KUKA KRL program: EPS_2_26115_ST7262_A_20260223020031.src

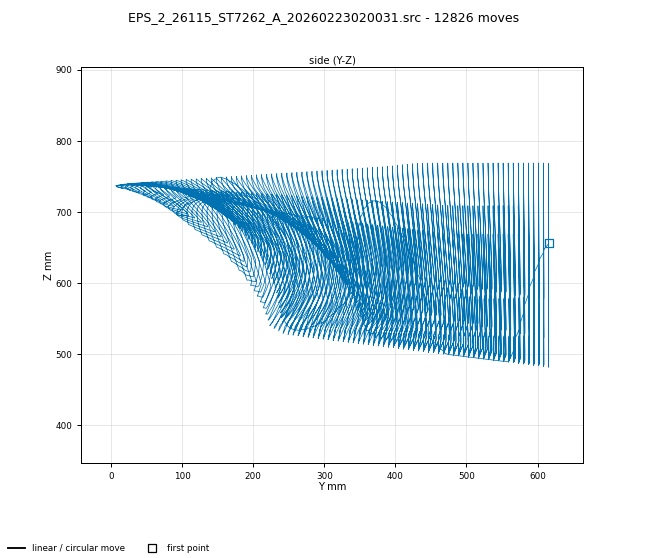
[picture p0: tool path of EPS_2_26115_ST7262_A_20260223020031.src, 12826 of 12828 moves have a stored position in this frame; points joined in program order, loops and branches not executed]
&ACCESS RVP
&REL 4
&COMMENT QRS 19112012
&PARAM EDITMASK = *
DEF PART()
EXT BAS (BAS_COMMAND :IN,REAL :IN )
INT I
BAS (#INITMOV,0 )

;KUKA QRS Post kuka4.cps  Date:22-06-2017 !

File_ID=3072

QRS_PRE_INIT()

;Init var - Until changes are made in qrs_pre_init
Outlet_Square_prg=0
Inlet_1_Square_prg=0
Inlet_2_Square_prg=0
Inlet_3_Square_prg=0
Inlet_4_Square_prg=0
Inlet_5_Square_prg=0

Outlet_1={X 0.000, Y 435.000, Z 586.000, B 0.000, E1 0.000 }
Inlet_1={X 0.000, Y 481.370, Z 486.000, B 0.000, E1 90.000 }
Inlet_2={X 0.000, Y 478.250, Z 526.000, B 0.000, E1 195.000 }
Outlet_1_type=366
Inlet_1_type=366
Inlet_2_type=366
;QRS#1=Sidecore dimensions
;QRS#2=375-15" PVC SDR 35 Cut Back
;QRS#3=375-15" PVC SDR 35
;QRS#4=375-15" PVC SDR 35
;QRS#5=
;QRS#6=
;QRS#7=
;QRS#8=
;QRS#9=20Y PSX
;QRS#10=20Y PSX
;QRS#11=20Y PSX
;QRS#12=
;QRS#13=
;QRS#14=
;QRS#15=
;QRS#16=1220x127x1067 3,5'
;QRS#17=EPS Height
;QRS#18=769
;QRS#19=*
;QRS#20= UPDATED VERSION 22-06-2017
;QRS#21=*
Outlet_Square=0250
Inlet_1_Square=0250
Inlet_2_Square=0250
Inlet_3_Square=0
Inlet_4_Square=0
Inlet_5_Square=0
Mill_Square=1
Outlet_Square_Prg=275
Inlet_1_Square_prg=252
Inlet_2_Square_prg=252

QRS_INIT()

$ADVANCE=5

; T1
PTP {E1 173.417,E2 173.417}
PTP {X 0,Y 615.494,A -85,B 0,C 180,E1 173.417,E2 173.417,E3 0,E4 0,E5 0,E6 0}
QRS_SPEED_INIT()
LIN {X 0,Y 615.494,Z 656.327,A -85,B 0,C 180,E1 173.417,E2 173.417,E3 0,E4 0,E5 0,E6 0} C_VEL
LIN {X 0,Y 615.488,Z 650.936,A -85,B 0,C 180,E1 172.124,E2 172.124} C_VEL
LIN {X 0,Y 615.489,Z 644.145,A -85,B 0,C 180,E1 170.801,E2 170.801} C_VEL
LIN {X 0,Y 615.492,Z 635.981,A -85,B 0,C 180,E1 169.473,E2 169.473} C_VEL
LIN {X 0,Y 615.494,Z 626.246,A -85,B 0,C 180,E1 168.139,E2 168.139} C_VEL
LIN {X 0,Y 615.49,Z 616.219,A -85,B 0,C 180,E1 166.966,E2 166.966} C_VEL
LIN {X 0,Y 615.496,Z 604.053,A -85,B 0,C 180,E1 165.759,E2 165.759} C_VEL
LIN {X 0,Y 615.5,Z 590.268,A -85,B 0,C 180,E1 164.604,E2 164.604} C_VEL
LIN {X 0,Y 615.495,Z 575.471,A -85,B 0,C 180,E1 163.567,E2 163.567} C_VEL
LIN {X 0,Y 615.499,Z 561.122,A -85,B 0,C 180,E1 162.73,E2 162.73} C_VEL
LIN {X 0,Y 615.48,Z 547.09,A -85,B 0,C 180,E1 162.043,E2 162.043} C_VEL
LIN {X 0,Y 615.499,Z 531.957,A -85,B 0,C 180,E1 161.434,E2 161.434} C_VEL
LIN {X 0,Y 615.48,Z 515.455,A -85,B 0,C 180,E1 160.921,E2 160.921} C_VEL
LIN {X 0,Y 615.494,Z 498.994,A -85,B 0,C 180,E1 160.554,E2 160.554} C_VEL
LIN {X 0,Y 615.49,Z 482.974,A -85,B 0,C 180,E1 160.315,E2 160.315} C_VEL
LIN {X 0,Y 615.487,Z 482.007,A -85,B 0,C 180,E1 159.269,E2 159.269} C_VEL
LIN {X 0,Y 615.491,Z 482.006,A -85,B 0,C 180,E1 156.443,E2 156.443} C_VEL
LIN {X 0,Y 615.479,Z 482.009,A -85,B 0,C 180,E1 153.555,E2 153.555} C_VEL
LIN {X 0,Y 615.491,Z 482.009,A -85,B 0,C 180,E1 151.342,E2 151.342} C_VEL
LIN {X 0,Y 615.477,Z 482.007,A -85,B 0,C 180,E1 148.916,E2 148.916} C_VEL
LIN {X 0,Y 615.494,Z 482.006,A -85,B 0,C 180,E1 146.465,E2 146.465} C_VEL
LIN {X 0,Y 615.481,Z 482.008,A -85,B 0,C 180,E1 143.574,E2 143.574} C_VEL
LIN {X 0,Y 615.49,Z 482.011,A -85,B 0,C 180,E1 140.938,E2 140.938} C_VEL
LIN {X 0,Y 615.482,Z 482.01,A -85,B 0,C 180,E1 138.525,E2 138.525} C_VEL
LIN {X 0,Y 615.482,Z 482.007,A -85,B 0,C 180,E1 135.849,E2 135.849} C_VEL
LIN {X 0,Y 615.485,Z 482.006,A -85,B 0,C 180,E1 133.047,E2 133.047} C_VEL
LIN {X 0,Y 615.495,Z 482.005,A -85,B 0,C 180,E1 130.089,E2 130.089} C_VEL
LIN {X 0,Y 615.49,Z 482.006,A -85,B 0,C 180,E1 127.242,E2 127.242} C_VEL
LIN {X 0,Y 615.477,Z 482.007,A -85,B 0,C 180,E1 124.698,E2 124.698} C_VEL
LIN {X 0,Y 615.497,Z 482.008,A -85,B 0,C 180,E1 122.332,E2 122.332} C_VEL
LIN {X 0,Y 615.485,Z 482.01,A -85,B 0,C 180,E1 119.407,E2 119.407} C_VEL
LIN {X 0,Y 615.492,Z 482.008,A -85,B 0,C 180,E1 117.045,E2 117.045} C_VEL
LIN {X 0,Y 615.498,Z 482.03,A -85,B 0,C 180,E1 114.141,E2 114.141} C_VEL
LIN {X 0,Y 615.499,Z 487.086,A -85,B 0,C 180,E1 111.432,E2 111.432} C_VEL
LIN {X 0,Y 615.477,Z 492.467,A -85,B 0,C 180,E1 108.6,E2 108.6} C_VEL
LIN {X 0,Y 615.494,Z 497.748,A -85,B 0,C 180,E1 105.906,E2 105.906} C_VEL
LIN {X 0,Y 615.487,Z 503.194,A -85,B 0,C 180,E1 103.202,E2 103.202} C_VEL
LIN {X 0,Y 615.476,Z 508.733,A -85,B 0,C 180,E1 100.528,E2 100.528} C_VEL
LIN {X 0,Y 615.487,Z 514.32,A -85,B 0,C 180,E1 97.876,E2 97.876} C_VEL
LIN {X 0,Y 615.491,Z 520.717,A -85,B 0,C 180,E1 94.913,E2 94.913} C_VEL
LIN {X 0,Y 615.481,Z 521.339,A -85,B 0,C 180,E1 94.626,E2 94.626} C_VEL
LIN {X 0,Y 615.497,Z 540.982,A -85,B 0,C 180,E1 94.319,E2 94.319} C_VEL
LIN {X 0,Y 615.486,Z 557.536,A -85,B 0,C 180,E1 93.929,E2 93.929} C_VEL
LIN {X 0,Y 615.475,Z 573.048,A -85,B 0,C 180,E1 93.438,E2 93.438} C_VEL
LIN {X 0,Y 615.487,Z 589.037,A -85,B 0,C 180,E1 92.782,E2 92.782} C_VEL
LIN {X 0,Y 615.498,Z 603.591,A -85,B 0,C 180,E1 92.046,E2 92.046} C_VEL
LIN {X 0,Y 615.497,Z 618.433,A -85,B 0,C 180,E1 91.146,E2 91.146} C_VEL
LIN {X 0,Y 615.497,Z 632.037,A -85,B 0,C 180,E1 90.164,E2 90.164} C_VEL
LIN {X 0,Y 615.494,Z 643.706,A -85,B 0,C 180,E1 89.183,E2 89.183} C_VEL
LIN {X 0,Y 615.499,Z 655.309,A -85,B 0,C 180,E1 88.038,E2 88.038} C_VEL
LIN {X 0,Y 615.492,Z 666.597,A -85,B 0,C 180,E1 86.728,E2 86.728} C_VEL
LIN {X 0,Y 615.491,Z 676.122,A -85,B 0,C 180,E1 85.416,E2 85.416} C_VEL
LIN {X 0,Y 615.493,Z 684.181,A -85,B 0,C 180,E1 84.102,E2 84.102} C_VEL
LIN {X 0,Y 615.493,Z 690.938,A -85,B 0,C 180,E1 82.785,E2 82.785} C_VEL
LIN {X 0,Y 615.487,Z 696.437,A -85,B 0,C 180,E1 81.464,E2 81.464} C_VEL
LIN {X 0,Y 615.496,Z 700.913,A -85,B 0,C 180,E1 80.139,E2 80.139} C_VEL
LIN {X 0,Y 615.494,Z 704.24,A -85,B 0,C 180,E1 78.808,E2 78.808} C_VEL
LIN {X 0,Y 615.489,Z 706.639,A -85,B 0,C 180,E1 77.471,E2 77.471} C_VEL
LIN {X 0,Y 615.49,Z 708.009,A -85,B 0,C 180,E1 76.068,E2 76.068} C_VEL
LIN {X 0,Y 615.492,Z 708.351,A -85,B 0,C 180,E1 74.775,E2 74.775} C_VEL
LIN {X 0,Y 615.491,Z 707.707,A -85,B 0,C 180,E1 73.414,E2 73.414} C_VEL
LIN {X 0,Y 615.489,Z 706.012,A -85,B 0,C 180,E1 72.044,E2 72.044} C_VEL
LIN {X 0,Y 615.49,Z 703.29,A -85,B 0,C 180,E1 70.663,E2 70.663} C_VEL
LIN {X 0,Y 615.497,Z 698.197,A -85,B 0,C 180,E1 68.92,E2 68.92} C_VEL
LIN {X 0,Y 615.499,Z 692.193,A -85,B 0,C 180,E1 67.406,E2 67.406} C_VEL
LIN {X 0,Y 615.492,Z 685.183,A -85,B 0,C 180,E1 65.992,E2 65.992} C_VEL
LIN {X 0,Y 615.493,Z 677.649,A -85,B 0,C 180,E1 64.721,E2 64.721} C_VEL
LIN {X 0,Y 615.492,Z 668.374,A -85,B 0,C 180,E1 63.407,E2 63.407} C_VEL
LIN {X 0,Y 615.493,Z 658.93,A -85,B 0,C 180,E1 62.271,E2 62.271} C_VEL
LIN {X 0,Y 615.494,Z 648.24,A -85,B 0,C 180,E1 61.157,E2 61.157} C_VEL
LIN {X 0,Y 615.495,Z 636.643,A -85,B 0,C 180,E1 60.114,E2 60.114} C_VEL
LIN {X 0,Y 615.496,Z 623.154,A -85,B 0,C 180,E1 59.082,E2 59.082} C_VEL
LIN {X 0,Y 615.498,Z 610.049,A -85,B 0,C 180,E1 58.236,E2 58.236} C_VEL
LIN {X 0,Y 615.498,Z 595.659,A -85,B 0,C 180,E1 57.447,E2 57.447} C_VEL
LIN {X 0,Y 615.483,Z 580.647,A -85,B 0,C 180,E1 56.765,E2 56.765} C_VEL
LIN {X 0,Y 615.477,Z 565.676,A -85,B 0,C 180,E1 56.224,E2 56.224} C_VEL
LIN {X 0,Y 615.489,Z 551.02,A -85,B 0,C 180,E1 55.81,E2 55.81} C_VEL
LIN {X 0,Y 615.492,Z 535.775,A -85,B 0,C 180,E1 55.493,E2 55.493} C_VEL
LIN {X 0,Y 615.48,Z 521.345,A -85,B 0,C 180,E1 55.287,E2 55.287} C_VEL
LIN {X 0,Y 615.491,Z 515.876,A -85,B 0,C 180,E1 52.76,E2 52.76} C_VEL
LIN {X 0,Y 615.489,Z 509.829,A -85,B 0,C 180,E1 49.911,E2 49.911} C_VEL
LIN {X 0,Y 615.49,Z 505.13,A -85,B 0,C 180,E1 47.649,E2 47.649} C_VEL
LIN {X 0,Y 615.48,Z 499.601,A -85,B 0,C 180,E1 44.932,E2 44.932} C_VEL
LIN {X 0,Y 615.494,Z 493.965,A -85,B 0,C 180,E1 42.083,E2 42.083} C_VEL
LIN {X 0,Y 615.498,Z 489.481,A -85,B 0,C 180,E1 39.75,E2 39.75} C_VEL
LIN {X 0,Y 615.48,Z 484.243,A -85,B 0,C 180,E1 36.938,E2 36.938} C_VEL
LIN {X 0,Y 615.495,Z 482.008,A -85,B 0,C 180,E1 35.726,E2 35.726} C_VEL
LIN {X 0,Y 615.491,Z 482.014,A -85,B 0,C 180,E1 33.236,E2 33.236} C_VEL
LIN {X 0,Y 615.483,Z 482.009,A -85,B 0,C 180,E1 30.92,E2 30.92} C_VEL
LIN {X 0,Y 615.483,Z 482.007,A -85,B 0,C 180,E1 28.452,E2 28.452} C_VEL
LIN {X 0,Y 615.496,Z 482.005,A -85,B 0,C 180,E1 25.574,E2 25.574} C_VEL
LIN {X 0,Y 615.482,Z 482.008,A -85,B 0,C 180,E1 22.845,E2 22.845} C_VEL
LIN {X 0,Y 615.477,Z 482.01,A -85,B 0,C 180,E1 20.033,E2 20.033} C_VEL
LIN {X 0,Y 615.49,Z 482.008,A -85,B 0,C 180,E1 17.271,E2 17.271} C_VEL
LIN {X 0,Y 615.493,Z 482.008,A -85,B 0,C 180,E1 14.549,E2 14.549} C_VEL
LIN {X 0,Y 615.48,Z 482.01,A -85,B 0,C 180,E1 11.861,E2 11.861} C_VEL
LIN {X 0,Y 615.488,Z 482.008,A -85,B 0,C 180,E1 9.199,E2 9.199} C_VEL
LIN {X 0,Y 615.491,Z 482.006,A -85,B 0,C 180,E1 6.557,E2 6.557} C_VEL
LIN {X 0,Y 615.475,Z 482.009,A -85,B 0,C 180,E1 3.929,E2 3.929} C_VEL
LIN {X 0,Y 615.488,Z 482.005,A -85,B 0,C 180,E1 1.309,E2 1.309} C_VEL
LIN {X 0,Y 615.486,Z 482.006,A -85,B 0,C 180,E1 -1.308,E2 -1.308} C_VEL
LIN {X 0,Y 615.476,Z 482.009,A -85,B 0,C 180,E1 -3.928,E2 -3.928} C_VEL
LIN {X 0,Y 615.491,Z 482.006,A -85,B 0,C 180,E1 -6.593,E2 -6.593} C_VEL
LIN {X 0,Y 615.48,Z 482.009,A -85,B 0,C 180,E1 -9.199,E2 -9.199} C_VEL
LIN {X 0,Y 615.48,Z 482.01,A -85,B 0,C 180,E1 -11.861,E2 -11.861} C_VEL
LIN {X 0,Y 615.493,Z 482.008,A -85,B 0,C 180,E1 -14.549,E2 -14.549} C_VEL
LIN {X 0,Y 615.481,Z 482.01,A -85,B 0,C 180,E1 -17.27,E2 -17.27} C_VEL
LIN {X 0,Y 615.482,Z 482.009,A -85,B 0,C 180,E1 -20.033,E2 -20.033} C_VEL
LIN {X 0,Y 615.483,Z 482.008,A -85,B 0,C 180,E1 -22.844,E2 -22.844} C_VEL
LIN {X 0,Y 615.493,Z 482.005,A -85,B 0,C 180,E1 -25.715,E2 -25.715} C_VEL
LIN {X 0,Y 615.49,Z 482.005,A -85,B 0,C 180,E1 -28.658,E2 -28.658} C_VEL
LIN {X 0,Y 615.477,Z 482.008,A -85,B 0,C 180,E1 -31.087,E2 -31.087} C_VEL
LIN {X 0,Y 615.488,Z 482.009,A -85,B 0,C 180,E1 -33.536,E2 -33.536} C_VEL
LIN {X 0,Y 615.489,Z 482.007,A -85,B 0,C 180,E1 -36.424,E2 -36.424} C_VEL
LIN {X 0,Y 615.479,Z 482.01,A -85,B 0,C 180,E1 -39.063,E2 -39.063} C_VEL
LIN {X 0,Y 615.499,Z 482.012,A -85,B 0,C 180,E1 -41.473,E2 -41.473} C_VEL
LIN {X 0,Y 615.497,Z 482.013,A -85,B 0,C 180,E1 -44.148,E2 -44.148} C_VEL
LIN {X 0,Y 615.486,Z 482.013,A -85,B 0,C 180,E1 -46.952,E2 -46.952} C_VEL
LIN {X 0,Y 615.489,Z 482.01,A -85,B 0,C 180,E1 -49.395,E2 -49.395} C_VEL
LIN {X 0,Y 615.481,Z 482.123,A -85,B 0,C 180,E1 -50.508,E2 -50.508} C_VEL
LIN {X 0,Y 615.485,Z 493.267,A -85,B 0,C 180,E1 -53.063,E2 -53.063} C_VEL
LIN {X 0,Y 615.482,Z 504.895,A -85,B 0,C 180,E1 -55.641,E2 -55.641} C_VEL
LIN {X 0,Y 615.476,Z 517.347,A -85,B 0,C 180,E1 -58.315,E2 -58.315} C_VEL
LIN {X 0,Y 615.491,Z 530.061,A -85,B 0,C 180,E1 -60.97,E2 -60.97} C_VEL
LIN {X 0,Y 615.492,Z 544.583,A -85,B 0,C 180,E1 -63.922,E2 -63.922} C_VEL
LIN {X 0,Y 615.488,Z 559.093,A -85,B 0,C 180,E1 -66.801,E2 -66.801} C_VEL
LIN {X 0,Y 615.491,Z 574.038,A -85,B 0,C 180,E1 -69.706,E2 -69.706} C_VEL
LIN {X 0,Y 615.477,Z 576.988,A -85,B 0,C 180,E1 -70.272,E2 -70.272} C_VEL
LIN {X 0,Y 615.481,Z 600.112,A -85,B 0,C 180,E1 -70.62,E2 -70.62} C_VEL
LIN {X 0,Y 615.49,Z 616.959,A -85,B 0,C 180,E1 -71.009,E2 -71.009} C_VEL
LIN {X 0,Y 615.481,Z 633.051,A -85,B 0,C 180,E1 -71.518,E2 -71.518} C_VEL
LIN {X 0,Y 615.487,Z 650.013,A -85,B 0,C 180,E1 -72.216,E2 -72.216} C_VEL
LIN {X 0,Y 615.498,Z 665.019,A -85,B 0,C 180,E1 -72.988,E2 -72.988} C_VEL
LIN {X 0,Y 615.497,Z 678.752,A -85,B 0,C 180,E1 -73.831,E2 -73.831} C_VEL
LIN {X 0,Y 615.499,Z 692.9,A -85,B 0,C 180,E1 -74.86,E2 -74.86} C_VEL
LIN {X 0,Y 615.496,Z 705.179,A -85,B 0,C 180,E1 -75.911,E2 -75.911} C_VEL
LIN {X 0,Y 615.494,Z 717.33,A -85,B 0,C 180,E1 -77.136,E2 -77.136} C_VEL
LIN {X 0,Y 615.49,Z 728.541,A -85,B 0,C 180,E1 -78.474,E2 -78.474} C_VEL
LIN {X 0,Y 615.493,Z 737.921,A -85,B 0,C 180,E1 -79.807,E2 -79.807} C_VEL
LIN {X 0,Y 615.494,Z 745.711,A -85,B 0,C 180,E1 -81.133,E2 -81.133} C_VEL
LIN {X 0,Y 615.491,Z 752.215,A -85,B 0,C 180,E1 -82.455,E2 -82.455} C_VEL
LIN {X 0,Y 615.493,Z 757.492,A -85,B 0,C 180,E1 -83.773,E2 -83.773} C_VEL
LIN {X 0,Y 615.496,Z 760.742,A -85,B 0,C 180,E1 -84.76,E2 -84.76} C_VEL
LIN {X 0,Y 615.494,Z 764.078,A -85,B 0,C 180,E1 -86.072,E2 -86.072} C_VEL
LIN {X 0,Y 615.486,Z 766.505,A -85,B 0,C 180,E1 -87.383,E2 -87.383} C_VEL
LIN {X 0,Y 615.493,Z 767.87,A -85,B 0,C 180,E1 -88.692,E2 -88.692} C_VEL
LIN {X 0,Y 615.489,Z 768.39,A -85,B 0,C 180,E1 -90.001,E2 -90.001} C_VEL
LIN {X 0,Y 615.493,Z 767.869,A -85,B 0,C 180,E1 -91.309,E2 -91.309} C_VEL
LIN {X 0,Y 615.486,Z 766.503,A -85,B 0,C 180,E1 -92.619,E2 -92.619} C_VEL
LIN {X 0,Y 615.494,Z 764.075,A -85,B 0,C 180,E1 -93.929,E2 -93.929} C_VEL
LIN {X 0,Y 615.496,Z 760.738,A -85,B 0,C 180,E1 -95.242,E2 -95.242} C_VEL
LIN {X 0,Y 615.495,Z 754.98,A -85,B 0,C 180,E1 -96.898,E2 -96.898} C_VEL
LIN {X 0,Y 615.489,Z 747.498,A -85,B 0,C 180,E1 -98.537,E2 -98.537} C_VEL
LIN {X 0,Y 615.491,Z 738.961,A -85,B 0,C 180,E1 -100.029,E2 -100.029} C_VEL
LIN {X 0,Y 615.496,Z 729.762,A -85,B 0,C 180,E1 -101.36,E2 -101.36} C_VEL
LIN {X 0,Y 615.494,Z 720.286,A -85,B 0,C 180,E1 -102.531,E2 -102.531} C_VEL
LIN {X 0,Y 615.493,Z 709.208,A -85,B 0,C 180,E1 -103.706,E2 -103.706} C_VEL
LIN {X 0,Y 615.496,Z 697.108,A -85,B 0,C 180,E1 -104.803,E2 -104.803} C_VEL
LIN {X 0,Y 615.497,Z 682.701,A -85,B 0,C 180,E1 -105.905,E2 -105.905} C_VEL
LIN {X 0,Y 615.497,Z 668.005,A -85,B 0,C 180,E1 -106.843,E2 -106.843} C_VEL
LIN {X 0,Y 615.498,Z 653.499,A -85,B 0,C 180,E1 -107.614,E2 -107.614} C_VEL
LIN {X 0,Y 615.487,Z 638.297,A -85,B 0,C 180,E1 -108.28,E2 -108.28} C_VEL
LIN {X 0,Y 615.49,Z 622.975,A -85,B 0,C 180,E1 -108.819,E2 -108.819} C_VEL
LIN {X 0,Y 615.488,Z 606.497,A -85,B 0,C 180,E1 -109.252,E2 -109.252} C_VEL
LIN {X 0,Y 615.476,Z 590.893,A -85,B 0,C 180,E1 -109.534,E2 -109.534} C_VEL
LIN {X 0,Y 615.477,Z 576.981,A -85,B 0,C 180,E1 -109.729,E2 -109.729} C_VEL
LIN {X 0,Y 615.481,Z 563.459,A -85,B 0,C 180,E1 -112.345,E2 -112.345} C_VEL
LIN {X 0,Y 615.491,Z 550.019,A -85,B 0,C 180,E1 -114.992,E2 -114.992} C_VEL
LIN {X 0,Y 615.483,Z 535.501,A -85,B 0,C 180,E1 -117.916,E2 -117.916} C_VEL
LIN {X 0,Y 615.479,Z 522.788,A -85,B 0,C 180,E1 -120.54,E2 -120.54} C_VEL
LIN {X 0,Y 615.49,Z 510.074,A -85,B 0,C 180,E1 -123.236,E2 -123.236} C_VEL
LIN {X 0,Y 615.494,Z 496.874,A -85,B 0,C 180,E1 -126.128,E2 -126.128} C_VEL
LIN {X 0,Y 615.485,Z 484.646,A -85,B 0,C 180,E1 -128.905,E2 -128.905} C_VEL
LIN {X 0,Y 615.48,Z 482.003,A -85,B 0,C 180,E1 -129.536,E2 -129.536} C_VEL
LIN {X 0,Y 615.49,Z 481.999,A -85,B 0,C 180,E1 -132.353,E2 -132.353} C_VEL
LIN {X 0,Y 615.491,Z 482.006,A -85,B 0,C 180,E1 -135.068,E2 -135.068} C_VEL
LIN {X 0,Y 615.477,Z 481.999,A -85,B 0,C 180,E1 -137.921,E2 -137.921} C_VEL
LIN {X 0,Y 615.498,Z 482.002,A -85,B 0,C 180,E1 -140.251,E2 -140.251} C_VEL
LIN {X 0,Y 615.483,Z 482,A -85,B 0,C 180,E1 -143.064,E2 -143.064} C_VEL
LIN {X 0,Y 615.491,Z 481.995,A -85,B 0,C 180,E1 -145.299,E2 -145.299} C_VEL
LIN {X 0,Y 615.49,Z 482.013,A -85,B 0,C 180,E1 -148.315,E2 -148.315} C_VEL
LIN {X 0,Y 615.482,Z 482.003,A -85,B 0,C 180,E1 -150.594,E2 -150.594} C_VEL
LIN {X 0,Y 615.478,Z 481.998,A -85,B 0,C 180,E1 -152.957,E2 -152.957} C_VEL
LIN {X 0,Y 615.493,Z 482.007,A -85,B 0,C 180,E1 -155.729,E2 -155.729} C_VEL
LIN {X 0,Y 615.486,Z 481.998,A -85,B 0,C 180,E1 -158.568,E2 -158.568} C_VEL
LIN {X 0,Y 615.492,Z 482.003,A -85,B 0,C 180,E1 -159.442,E2 -159.442} C_VEL
LIN {X 0,Y 615.493,Z 482.97,A -85,B 0,C 180,E1 -160.402,E2 -160.402} C_VEL
LIN {X 0,Y 615.493,Z 501.134,A -85,B 0,C 180,E1 -160.684,E2 -160.684} C_VEL
LIN {X 0,Y 615.486,Z 516.875,A -85,B 0,C 180,E1 -161.052,E2 -161.052} C_VEL
LIN {X 0,Y 615.494,Z 532.859,A -85,B 0,C 180,E1 -161.556,E2 -161.556} C_VEL
LIN {X 0,Y 615.485,Z 547.011,A -85,B 0,C 180,E1 -162.129,E2 -162.129} C_VEL
LIN {X 0,Y 615.497,Z 562.619,A -85,B 0,C 180,E1 -162.901,E2 -162.901} C_VEL
LIN {X 0,Y 615.499,Z 576.095,A -85,B 0,C 180,E1 -163.698,E2 -163.698} C_VEL
LIN {X 0,Y 615.496,Z 590.21,A -85,B 0,C 180,E1 -164.69,E2 -164.69} C_VEL
LIN {X 0,Y 615.492,Z 603.031,A -85,B 0,C 180,E1 -165.758,E2 -165.758} C_VEL
LIN {X 0,Y 615.493,Z 613.734,A -85,B 0,C 180,E1 -166.799,E2 -166.799} C_VEL
LIN {X 0,Y 615.498,Z 624.165,A -85,B 0,C 180,E1 -167.973,E2 -167.973} C_VEL
LIN {X 0,Y 615.492,Z 632.908,A -85,B 0,C 180,E1 -169.11,E2 -169.11} C_VEL
LIN {X 0,Y 615.498,Z 641.712,A -85,B 0,C 180,E1 -170.47,E2 -170.47} C_VEL
LIN {X 0,Y 615.491,Z 648.891,A -85,B 0,C 180,E1 -171.794,E2 -171.794} C_VEL
LIN {X 0,Y 615.494,Z 654.786,A -85,B 0,C 180,E1 -173.1,E2 -173.1} C_VEL
LIN {X 0,Y 615.495,Z 660.597,A -85,B 0,C 180,E1 -174.759,E2 -174.759} C_VEL
LIN {X 0,Y 615.489,Z 663.98,A -85,B 0,C 180,E1 -176.072,E2 -176.072} C_VEL
LIN {X 0,Y 615.496,Z 666.428,A -85,B 0,C 180,E1 -177.382,E2 -177.382} C_VEL
LIN {X 0,Y 615.489,Z 667.838,A -85,B 0,C 180,E1 -178.692,E2 -178.692} C_VEL
LIN {X 0,Y 615.491,Z 668.385,A -85,B 0,C 180,E1 -180,E2 -180} C_VEL
LIN {X 0,Y 615.49,Z 667.901,A -85,B 0,C 180,E1 -181.309,E2 -181.309} C_VEL
LIN {X 0,Y 615.493,Z 666.567,A -85,B 0,C 180,E1 -182.618,E2 -182.618} C_VEL
LIN {X 0,Y 615.491,Z 664.174,A -85,B 0,C 180,E1 -183.929,E2 -183.929} C_VEL
LIN {X 0,Y 615.49,Z 660.878,A -85,B 0,C 180,E1 -185.241,E2 -185.241} C_VEL
LIN {X 0,Y 615.494,Z 656.327,A -85,B 0,C 180,E1 -186.583,E2 -186.583} C_VEL
LIN {X 0,Y 614.816,Z 654.479,A -85,B 0,C 180,E1 -187.099,E2 -187.099} C_VEL
LIN {X 0,Y 611.953,Z 651.273,A -85,B 0,C 180,E1 -187.93,E2 -187.93} C_VEL
LIN {X 0,Y 609.092,Z 647.426,A -85,B 0,C 180,E1 -188.752,E2 -188.752} C_VEL
LIN {X 0,Y 608.437,Z 644.768,A -85,B 0,C 180,E1 -189.252,E2 -189.252} C_VEL
LIN {X 0,Y 608.45,Z 636.228,A -85,B 0,C 180,E1 -190.65,E2 -190.65} C_VEL
LIN {X 0,Y 608.475,Z 626.412,A -85,B 0,C 180,E1 -192,E2 -192} C_VEL
LIN {X 0,Y 608.489,Z 616.317,A -85,B 0,C 180,E1 -193.186,E2 -193.186} C_VEL
LIN {X 0,Y 608.532,Z 604.419,A -85,B 0,C 180,E1 -194.378,E2 -194.378} C_VEL
LIN {X 0,Y 608.553,Z 591.342,A -85,B 0,C 180,E1 -195.49,E2 -195.49} C_VEL
LIN {X 0,Y 608.591,Z 578.47,A -85,B 0,C 180,E1 -196.422,E2 -196.422} C_VEL
LIN {X 0,Y 608.656,Z 564.25,A -85,B 0,C 180,E1 -197.298,E2 -197.298} C_VEL
LIN {X 0,Y 608.67,Z 549.051,A -85,B 0,C 180,E1 -198.078,E2 -198.078} C_VEL
LIN {X 0,Y 608.727,Z 533.997,A -85,B 0,C 180,E1 -198.703,E2 -198.703} C_VEL
LIN {X 0,Y 608.74,Z 518.47,A -85,B 0,C 180,E1 -199.211,E2 -199.211} C_VEL
LIN {X 0,Y 608.797,Z 502.403,A -85,B 0,C 180,E1 -199.603,E2 -199.603} C_VEL
LIN {X 0,Y 608.625,Z 484.542,A -85,B 0,C 180,E1 -199.896,E2 -199.896} C_VEL
LIN {X 0,Y 608.428,Z 483.38,A -85,B 0,C 180,E1 -199.923,E2 -199.923} C_VEL
LIN {X 0,Y 608.472,Z 483.004,A -85,B 0,C 180,E1 -200.68,E2 -200.68} C_VEL
LIN {X 0,Y 608.452,Z 483.01,A -85,B 0,C 180,E1 -203.124,E2 -203.124} C_VEL
LIN {X 0,Y 608.48,Z 483.004,A -85,B 0,C 180,E1 -205.722,E2 -205.722} C_VEL
LIN {X 0,Y 608.475,Z 483.004,A -85,B 0,C 180,E1 -208.62,E2 -208.62} C_VEL
LIN {X 0,Y 608.448,Z 483.007,A -85,B 0,C 180,E1 -211.318,E2 -211.318} C_VEL
LIN {X 0,Y 608.476,Z 483.002,A -85,B 0,C 180,E1 -213.735,E2 -213.735} C_VEL
LIN {X 0,Y 608.481,Z 483.007,A -85,B 0,C 180,E1 -216.09,E2 -216.09} C_VEL
LIN {X 0,Y 608.445,Z 483.008,A -85,B 0,C 180,E1 -218.59,E2 -218.59} C_VEL
LIN {X 0,Y 608.457,Z 483.005,A -85,B 0,C 180,E1 -221.341,E2 -221.341} C_VEL
LIN {X 0,Y 608.472,Z 483.003,A -85,B 0,C 180,E1 -223.87,E2 -223.87} C_VEL
LIN {X 0,Y 608.486,Z 483.001,A -85,B 0,C 180,E1 -226.69,E2 -226.69} C_VEL
LIN {X 0,Y 608.457,Z 483.005,A -85,B 0,C 180,E1 -229.697,E2 -229.697} C_VEL
LIN {X 0,Y 608.47,Z 483.004,A -85,B 0,C 180,E1 -232.253,E2 -232.253} C_VEL
LIN {X 0,Y 608.444,Z 483.007,A -85,B 0,C 180,E1 -235.096,E2 -235.096} C_VEL
LIN {X 0,Y 608.469,Z 483.009,A -85,B 0,C 180,E1 -237.477,E2 -237.477} C_VEL
LIN {X 0,Y 608.478,Z 483.006,A -85,B 0,C 180,E1 -240.221,E2 -240.221} C_VEL
LIN {X 0,Y 608.455,Z 483.01,A -85,B 0,C 180,E1 -243.226,E2 -243.226} C_VEL
LIN {X 0,Y 608.482,Z 483.122,A -85,B 0,C 180,E1 -245.926,E2 -245.926} C_VEL
LIN {X 0,Y 608.48,Z 487.635,A -85,B 0,C 180,E1 -248.308,E2 -248.308} C_VEL
LIN {X 0,Y 608.468,Z 493.236,A -85,B 0,C 180,E1 -251.286,E2 -251.286} C_VEL
LIN {X 0,Y 608.446,Z 498.329,A -85,B 0,C 180,E1 -253.905,E2 -253.905} C_VEL
LIN {X 0,Y 608.466,Z 503.8,A -85,B 0,C 180,E1 -256.643,E2 -256.643} C_VEL
LIN {X 0,Y 608.43,Z 509.353,A -85,B 0,C 180,E1 -259.349,E2 -259.349} C_VEL
LIN {X 0,Y 608.446,Z 514.98,A -85,B 0,C 180,E1 -262.032,E2 -262.032} C_VEL
LIN {X 0,Y 608.444,Z 520.684,A -85,B 0,C 180,E1 -264.697,E2 -264.697} C_VEL
LIN {X 0,Y 608.458,Z 521.747,A -85,B 0,C 180,E1 -265.154,E2 -265.154} C_VEL
LIN {X 0,Y 608.795,Z 524.408,A -85,B 0,C 180,E1 -265.198,E2 -265.198} C_VEL
LIN {X 0,Y 608.811,Z 541.409,A -85,B 0,C 180,E1 -265.468,E2 -265.468} C_VEL
LIN {X 0,Y 608.76,Z 557.825,A -85,B 0,C 180,E1 -265.862,E2 -265.862} C_VEL
LIN {X 0,Y 608.711,Z 573.288,A -85,B 0,C 180,E1 -266.359,E2 -266.359} C_VEL
LIN {X 0,Y 608.696,Z 589.244,A -85,B 0,C 180,E1 -267.021,E2 -267.021} C_VEL
LIN {X 0,Y 608.639,Z 603.778,A -85,B 0,C 180,E1 -267.766,E2 -267.766} C_VEL
LIN {X 0,Y 608.6,Z 618.584,A -85,B 0,C 180,E1 -268.676,E2 -268.676} C_VEL
LIN {X 0,Y 608.554,Z 632.189,A -85,B 0,C 180,E1 -269.668,E2 -269.668} C_VEL
LIN {X 0,Y 608.531,Z 643.867,A -85,B 0,C 180,E1 -270.661,E2 -270.661} C_VEL
LIN {X 0,Y 608.494,Z 655.51,A -85,B 0,C 180,E1 -271.819,E2 -271.819} C_VEL
LIN {X 0,Y 608.487,Z 666.842,A -85,B 0,C 180,E1 -273.144,E2 -273.144} C_VEL
LIN {X 0,Y 608.449,Z 676.437,A -85,B 0,C 180,E1 -274.471,E2 -274.471} C_VEL
LIN {X 0,Y 608.464,Z 683.653,A -85,B 0,C 180,E1 -275.633,E2 -275.633} C_VEL
LIN {X 0,Y 608.441,Z 690.561,A -85,B 0,C 180,E1 -276.965,E2 -276.965} C_VEL
LIN {X 0,Y 608.451,Z 696.303,A -85,B 0,C 180,E1 -278.301,E2 -278.301} C_VEL
LIN {X 0,Y 608.424,Z 700.921,A -85,B 0,C 180,E1 -279.641,E2 -279.641} C_VEL
LIN {X 0,Y 608.421,Z 704.328,A -85,B 0,C 180,E1 -280.93,E2 -280.93} C_VEL
LIN {X 0,Y 608.436,Z 706.423,A -85,B 0,C 180,E1 -281.999,E2 -281.999} C_VEL
LIN {X 0,Y 608.429,Z 708.219,A -85,B 0,C 180,E1 -283.356,E2 -283.356} C_VEL
LIN {X 0,Y 608.409,Z 708.93,A -85,B 0,C 180,E1 -284.721,E2 -284.721} C_VEL
LIN {X 0,Y 608.414,Z 708.671,A -85,B 0,C 180,E1 -286.094,E2 -286.094} C_VEL
LIN {X 0,Y 608.417,Z 707.362,A -85,B 0,C 180,E1 -287.477,E2 -287.477} C_VEL
LIN {X 0,Y 608.423,Z 704.957,A -85,B 0,C 180,E1 -288.87,E2 -288.87} C_VEL
LIN {X 0,Y 608.435,Z 701.469,A -85,B 0,C 180,E1 -290.274,E2 -290.274} C_VEL
LIN {X 0,Y 608.424,Z 696.665,A -85,B 0,C 180,E1 -291.692,E2 -291.692} C_VEL
LIN {X 0,Y 608.448,Z 690.569,A -85,B 0,C 180,E1 -293.123,E2 -293.123} C_VEL
LIN {X 0,Y 608.469,Z 682.989,A -85,B 0,C 180,E1 -294.569,E2 -294.569} C_VEL
LIN {X 0,Y 608.455,Z 675.093,A -85,B 0,C 180,E1 -295.821,E2 -295.821} C_VEL
LIN {X 0,Y 608.499,Z 665.789,A -85,B 0,C 180,E1 -297.076,E2 -297.076} C_VEL
LIN {X 0,Y 608.495,Z 655.58,A -85,B 0,C 180,E1 -298.263,E2 -298.263} C_VEL
LIN {X 0,Y 608.519,Z 644.235,A -85,B 0,C 180,E1 -299.395,E2 -299.395} C_VEL
LIN {X 0,Y 608.575,Z 630.746,A -85,B 0,C 180,E1 -300.538,E2 -300.538} C_VEL
LIN {X 0,Y 608.617,Z 617.298,A -85,B 0,C 180,E1 -301.5,E2 -301.5} C_VEL
LIN {X 0,Y 608.656,Z 603.695,A -85,B 0,C 180,E1 -302.328,E2 -302.328} C_VEL
LIN {X 0,Y 608.687,Z 588.305,A -85,B 0,C 180,E1 -303.111,E2 -303.111} C_VEL
LIN {X 0,Y 608.724,Z 572.233,A -85,B 0,C 180,E1 -303.77,E2 -303.77} C_VEL
LIN {X 0,Y 608.756,Z 556.252,A -85,B 0,C 180,E1 -304.274,E2 -304.274} C_VEL
LIN {X 0,Y 608.803,Z 540.506,A -85,B 0,C 180,E1 -304.64,E2 -304.64} C_VEL
LIN {X 0,Y 608.762,Z 523.211,A -85,B 0,C 180,E1 -304.907,E2 -304.907} C_VEL
LIN {X 0,Y 608.437,Z 521.64,A -85,B 0,C 180,E1 -304.951,E2 -304.951} C_VEL
LIN {X 0,Y 608.425,Z 515.64,A -85,B 0,C 180,E1 -307.748,E2 -307.748} C_VEL
LIN {X 0,Y 608.432,Z 510.215,A -85,B 0,C 180,E1 -310.326,E2 -310.326} C_VEL
LIN {X 0,Y 608.448,Z 504.793,A -85,B 0,C 180,E1 -312.959,E2 -312.959} C_VEL
LIN {X 0,Y 608.463,Z 499.218,A -85,B 0,C 180,E1 -315.734,E2 -315.734} C_VEL
LIN {X 0,Y 608.456,Z 493.52,A -85,B 0,C 180,E1 -318.657,E2 -318.657} C_VEL
LIN {X 0,Y 608.465,Z 488.322,A -85,B 0,C 180,E1 -321.411,E2 -321.411} C_VEL
LIN {X 0,Y 608.477,Z 483.541,A -85,B 0,C 180,E1 -323.949,E2 -323.949} C_VEL
LIN {X 0,Y 608.478,Z 483.004,A -85,B 0,C 180,E1 -324.337,E2 -324.337} C_VEL
LIN {X 0,Y 608.458,Z 483.006,A -85,B 0,C 180,E1 -327.12,E2 -327.12} C_VEL
LIN {X 0,Y 608.466,Z 483.009,A -85,B 0,C 180,E1 -329.455,E2 -329.455} C_VEL
LIN {X 0,Y 608.45,Z 483.007,A -85,B 0,C 180,E1 -331.733,E2 -331.733} C_VEL
LIN {X 0,Y 608.477,Z 483.003,A -85,B 0,C 180,E1 -334.275,E2 -334.275} C_VEL
LIN {X 0,Y 608.449,Z 483.006,A -85,B 0,C 180,E1 -336.876,E2 -336.876} C_VEL
LIN {X 0,Y 608.464,Z 483.005,A -85,B 0,C 180,E1 -339.319,E2 -339.319} C_VEL
LIN {X 0,Y 608.453,Z 483.009,A -85,B 0,C 180,E1 -341.828,E2 -341.828} C_VEL
LIN {X 0,Y 608.463,Z 483.007,A -85,B 0,C 180,E1 -344.594,E2 -344.594} C_VEL
LIN {X 0,Y 608.479,Z 483.005,A -85,B 0,C 180,E1 -347.323,E2 -347.323} C_VEL
LIN {X 0,Y 608.459,Z 483.007,A -85,B 0,C 180,E1 -350.022,E2 -350.022} C_VEL
LIN {X 0,Y 608.476,Z 483.006,A -85,B 0,C 180,E1 -352.7,E2 -352.7} C_VEL
LIN {X 0,Y 608.466,Z 483.008,A -85,B 0,C 180,E1 -355.362,E2 -355.362} C_VEL
LIN {X 0,Y 608.466,Z 483.008,A -85,B 0,C 180,E1 -358.014,E2 -358.014} C_VEL
LIN {X 0,Y 608.484,Z 483.007,A -85,B 0,C 180,E1 -360.661,E2 -360.661} C_VEL
LIN {X 0,Y 608.478,Z 483.007,A -85,B 0,C 180,E1 -363.31,E2 -363.31} C_VEL
LIN {X 0,Y 608.454,Z 483.008,A -85,B 0,C 180,E1 -365.967,E2 -365.967} C_VEL
LIN {X 0,Y 608.458,Z 483.008,A -85,B 0,C 180,E1 -368.636,E2 -368.636} C_VEL
LIN {X 0,Y 608.468,Z 483.006,A -85,B 0,C 180,E1 -371.324,E2 -371.324} C_VEL
LIN {X 0,Y 608.457,Z 483.007,A -85,B 0,C 180,E1 -374.037,E2 -374.037} C_VEL
LIN {X 0,Y 608.473,Z 483.005,A -85,B 0,C 180,E1 -376.783,E2 -376.783} C_VEL
LIN {X 0,Y 608.446,Z 483.01,A -85,B 0,C 180,E1 -379.57,E2 -379.57} C_VEL
LIN {X 0,Y 608.483,Z 483.006,A -85,B 0,C 180,E1 -382.485,E2 -382.485} C_VEL
LIN {X 0,Y 608.458,Z 483.008,A -85,B 0,C 180,E1 -385.3,E2 -385.3} C_VEL
LIN {X 0,Y 608.446,Z 483.008,A -85,B 0,C 180,E1 -387.518,E2 -387.518} C_VEL
LIN {X 0,Y 608.465,Z 483.004,A -85,B 0,C 180,E1 -389.974,E2 -389.974} C_VEL
LIN {X 0,Y 608.462,Z 483.005,A -85,B 0,C 180,E1 -392.525,E2 -392.525} C_VEL
LIN {X 0,Y 608.449,Z 483.006,A -85,B 0,C 180,E1 -395.277,E2 -395.277} C_VEL
LIN {X 0,Y 608.466,Z 483.005,A -85,B 0,C 180,E1 -397.746,E2 -397.746} C_VEL
LIN {X 0,Y 608.472,Z 483.005,A -85,B 0,C 180,E1 -400.333,E2 -400.333} C_VEL
LIN {X 0,Y 608.466,Z 483.004,A -85,B 0,C 180,E1 -403.31,E2 -403.31} C_VEL
LIN {X 0,Y 608.469,Z 483.004,A -85,B 0,C 180,E1 -406.132,E2 -406.132} C_VEL
LIN {X 0,Y 608.459,Z 483.006,A -85,B 0,C 180,E1 -408.825,E2 -408.825} C_VEL
LIN {X 0,Y 608.484,Z 483.065,A -85,B 0,C 180,E1 -410.187,E2 -410.187} C_VEL
LIN {X 0,Y 608.692,Z 486.676,A -85,B 0,C 180,E1 -411.054,E2 -411.054} C_VEL
LIN {X 0,Y 608.68,Z 497.368,A -85,B 0,C 180,E1 -413.515,E2 -413.515} C_VEL
LIN {X 0,Y 608.641,Z 510.082,A -85,B 0,C 180,E1 -416.342,E2 -416.342} C_VEL
LIN {X 0,Y 608.583,Z 522.831,A -85,B 0,C 180,E1 -419.085,E2 -419.085} C_VEL
LIN {X 0,Y 608.564,Z 535.51,A -85,B 0,C 180,E1 -421.74,E2 -421.74} C_VEL
LIN {X 0,Y 608.549,Z 548.95,A -85,B 0,C 180,E1 -424.485,E2 -424.485} C_VEL
LIN {X 0,Y 608.5,Z 562.756,A -85,B 0,C 180,E1 -427.239,E2 -427.239} C_VEL
LIN {X 0,Y 608.501,Z 577.057,A -85,B 0,C 180,E1 -430.037,E2 -430.037} C_VEL
LIN {X 0,Y 608.815,Z 579.294,A -85,B 0,C 180,E1 -430.091,E2 -430.091} C_VEL
LIN {X 0,Y 608.775,Z 598.972,A -85,B 0,C 180,E1 -430.375,E2 -430.375} C_VEL
LIN {X 0,Y 608.754,Z 615.443,A -85,B 0,C 180,E1 -430.747,E2 -430.747} C_VEL
LIN {X 0,Y 608.724,Z 631.936,A -85,B 0,C 180,E1 -431.264,E2 -431.264} C_VEL
LIN {X 0,Y 608.672,Z 648.058,A -85,B 0,C 180,E1 -431.923,E2 -431.923} C_VEL
LIN {X 0,Y 608.655,Z 663.455,A -85,B 0,C 180,E1 -432.704,E2 -432.704} C_VEL
LIN {X 0,Y 608.593,Z 677.774,A -85,B 0,C 180,E1 -433.576,E2 -433.576} C_VEL
LIN {X 0,Y 608.556,Z 690.801,A -85,B 0,C 180,E1 -434.511,E2 -434.511} C_VEL
LIN {X 0,Y 608.548,Z 703.95,A -85,B 0,C 180,E1 -435.624,E2 -435.624} C_VEL
LIN {X 0,Y 608.504,Z 715.898,A -85,B 0,C 180,E1 -436.815,E2 -436.815} C_VEL
LIN {X 0,Y 608.475,Z 726.059,A -85,B 0,C 180,E1 -438.001,E2 -438.001} C_VEL
LIN {X 0,Y 608.45,Z 735.934,A -85,B 0,C 180,E1 -439.351,E2 -439.351} C_VEL
LIN {X 0,Y 608.438,Z 744.232,A -85,B 0,C 180,E1 -440.695,E2 -440.695} C_VEL
LIN {X 0,Y 608.453,Z 751.107,A -85,B 0,C 180,E1 -442.034,E2 -442.034} C_VEL
LIN {X 0,Y 608.437,Z 756.841,A -85,B 0,C 180,E1 -443.4,E2 -443.4} C_VEL
LIN {X 0,Y 608.438,Z 761.248,A -85,B 0,C 180,E1 -444.699,E2 -444.699} C_VEL
LIN {X 0,Y 608.431,Z 764.634,A -85,B 0,C 180,E1 -446.027,E2 -446.027} C_VEL
LIN {X 0,Y 608.413,Z 767.087,A -85,B 0,C 180,E1 -447.352,E2 -447.352} C_VEL
LIN {X 0,Y 608.445,Z 768.477,A -85,B 0,C 180,E1 -448.677,E2 -448.677} C_VEL
LIN {X 0,Y 608.429,Z 769,A -85,B 0,C 180,E1 -450.001,E2 -450.001} C_VEL
LIN {X 0,Y 608.445,Z 768.476,A -85,B 0,C 180,E1 -451.324,E2 -451.324} C_VEL
LIN {X 0,Y 608.413,Z 767.085,A -85,B 0,C 180,E1 -452.649,E2 -452.649} C_VEL
LIN {X 0,Y 608.431,Z 764.631,A -85,B 0,C 180,E1 -453.975,E2 -453.975} C_VEL
LIN {X 0,Y 608.438,Z 761.243,A -85,B 0,C 180,E1 -455.303,E2 -455.303} C_VEL
LIN {X 0,Y 608.44,Z 755.466,A -85,B 0,C 180,E1 -456.967,E2 -456.967} C_VEL
LIN {X 0,Y 608.444,Z 747.854,A -85,B 0,C 180,E1 -458.637,E2 -458.637} C_VEL
LIN {X 0,Y 608.458,Z 739.241,A -85,B 0,C 180,E1 -460.146,E2 -460.146} C_VEL
LIN {X 0,Y 608.465,Z 729.963,A -85,B 0,C 180,E1 -461.493,E2 -461.493} C_VEL
LIN {X 0,Y 608.491,Z 720.416,A -85,B 0,C 180,E1 -462.677,E2 -462.677} C_VEL
LIN {X 0,Y 608.519,Z 708.972,A -85,B 0,C 180,E1 -463.896,E2 -463.896} C_VEL
LIN {X 0,Y 608.555,Z 697.136,A -85,B 0,C 180,E1 -464.976,E2 -464.976} C_VEL
LIN {X 0,Y 608.607,Z 682.703,A -85,B 0,C 180,E1 -466.09,E2 -466.09} C_VEL
LIN {X 0,Y 608.623,Z 668.007,A -85,B 0,C 180,E1 -467.039,E2 -467.039} C_VEL
LIN {X 0,Y 608.681,Z 653.501,A -85,B 0,C 180,E1 -467.817,E2 -467.817} C_VEL
LIN {X 0,Y 608.724,Z 638.298,A -85,B 0,C 180,E1 -468.491,E2 -468.491} C_VEL
LIN {X 0,Y 608.765,Z 622.976,A -85,B 0,C 180,E1 -469.035,E2 -469.035} C_VEL
LIN {X 0,Y 608.769,Z 606.498,A -85,B 0,C 180,E1 -469.473,E2 -469.473} C_VEL
LIN {X 0,Y 608.808,Z 590.893,A -85,B 0,C 180,E1 -469.757,E2 -469.757} C_VEL
LIN {X 0,Y 608.622,Z 577.829,A -85,B 0,C 180,E1 -469.933,E2 -469.933} C_VEL
LIN {X 0,Y 608.501,Z 577.049,A -85,B 0,C 180,E1 -469.965,E2 -469.965} C_VEL
LIN {X 0,Y 608.501,Z 562.748,A -85,B 0,C 180,E1 -472.763,E2 -472.763} C_VEL
LIN {X 0,Y 608.55,Z 548.945,A -85,B 0,C 180,E1 -475.516,E2 -475.516} C_VEL
LIN {X 0,Y 608.564,Z 535.502,A -85,B 0,C 180,E1 -478.261,E2 -478.261} C_VEL
LIN {X 0,Y 608.584,Z 522.824,A -85,B 0,C 180,E1 -480.916,E2 -480.916} C_VEL
LIN {X 0,Y 608.653,Z 509.611,A -85,B 0,C 180,E1 -483.761,E2 -483.761} C_VEL
LIN {X 0,Y 608.684,Z 497.36,A -85,B 0,C 180,E1 -486.487,E2 -486.487} C_VEL
LIN {X 0,Y 608.713,Z 485.052,A -85,B 0,C 180,E1 -489.326,E2 -489.326} C_VEL
LIN {X 0,Y 608.451,Z 483.004,A -85,B 0,C 180,E1 -489.871,E2 -489.871} C_VEL
LIN {X 0,Y 608.462,Z 483.001,A -85,B 0,C 180,E1 -492.335,E2 -492.335} C_VEL
LIN {X 0,Y 608.461,Z 483.01,A -85,B 0,C 180,E1 -494.796,E2 -494.796} C_VEL
LIN {X 0,Y 608.458,Z 483.005,A -85,B 0,C 180,E1 -497.041,E2 -497.041} C_VEL
LIN {X 0,Y 608.453,Z 483.001,A -85,B 0,C 180,E1 -499.697,E2 -499.697} C_VEL
LIN {X 0,Y 608.465,Z 483.005,A -85,B 0,C 180,E1 -502.254,E2 -502.254} C_VEL
LIN {X 0,Y 608.483,Z 482.998,A -85,B 0,C 180,E1 -505.09,E2 -505.09} C_VEL
LIN {X 0,Y 608.465,Z 483.003,A -85,B 0,C 180,E1 -507.906,E2 -507.906} C_VEL
LIN {X 0,Y 608.483,Z 483.006,A -85,B 0,C 180,E1 -510.222,E2 -510.222} C_VEL
LIN {X 0,Y 608.472,Z 482.999,A -85,B 0,C 180,E1 -512.794,E2 -512.794} C_VEL
LIN {X 0,Y 608.454,Z 483.003,A -85,B 0,C 180,E1 -515.429,E2 -515.429} C_VEL
LIN {X 0,Y 608.471,Z 483.001,A -85,B 0,C 180,E1 -518.309,E2 -518.309} C_VEL
LIN {X 0,Y 608.432,Z 483.013,A -85,B 0,C 180,E1 -519.725,E2 -519.725} C_VEL
LIN {X 0,Y 608.436,Z 483.378,A -85,B 0,C 180,E1 -520.166,E2 -520.166} C_VEL
LIN {X 0,Y 608.828,Z 486.303,A -85,B 0,C 180,E1 -520.223,E2 -520.223} C_VEL
LIN {X 0,Y 608.808,Z 502.321,A -85,B 0,C 180,E1 -520.485,E2 -520.485} C_VEL
LIN {X 0,Y 608.763,Z 518.421,A -85,B 0,C 180,E1 -520.878,E2 -520.878} C_VEL
LIN {X 0,Y 608.72,Z 533.974,A -85,B 0,C 180,E1 -521.386,E2 -521.386} C_VEL
LIN {X 0,Y 608.679,Z 548.997,A -85,B 0,C 180,E1 -522.01,E2 -522.01} C_VEL
LIN {X 0,Y 608.639,Z 564.2,A -85,B 0,C 180,E1 -522.789,E2 -522.789} C_VEL
LIN {X 0,Y 608.603,Z 578.092,A -85,B 0,C 180,E1 -523.643,E2 -523.643} C_VEL
LIN {X 0,Y 608.549,Z 591.3,A -85,B 0,C 180,E1 -524.596,E2 -524.596} C_VEL
LIN {X 0,Y 608.531,Z 603.44,A -85,B 0,C 180,E1 -525.623,E2 -525.623} C_VEL
LIN {X 0,Y 608.504,Z 615.463,A -85,B 0,C 180,E1 -526.815,E2 -526.815} C_VEL
LIN {X 0,Y 608.477,Z 625.694,A -85,B 0,C 180,E1 -528.001,E2 -528.001} C_VEL
LIN {X 0,Y 608.455,Z 635.631,A -85,B 0,C 180,E1 -529.35,E2 -529.35} C_VEL
LIN {X 0,Y 608.441,Z 643.987,A -85,B 0,C 180,E1 -530.694,E2 -530.694} C_VEL
LIN {X 0,Y 608.449,Z 650.888,A -85,B 0,C 180,E1 -532.033,E2 -532.033} C_VEL
LIN {X 0,Y 608.444,Z 656.661,A -85,B 0,C 180,E1 -533.397,E2 -533.397} C_VEL
LIN {X 0,Y 608.439,Z 661.103,A -85,B 0,C 180,E1 -534.698,E2 -534.698} C_VEL
LIN {X 0,Y 608.427,Z 664.536,A -85,B 0,C 180,E1 -536.026,E2 -536.026} C_VEL
LIN {X 0,Y 608.423,Z 667.012,A -85,B 0,C 180,E1 -537.352,E2 -537.352} C_VEL
LIN {X 0,Y 608.442,Z 668.446,A -85,B 0,C 180,E1 -538.677,E2 -538.677} C_VEL
LIN {X 0,Y 608.432,Z 668.995,A -85,B 0,C 180,E1 -540,E2 -540} C_VEL
LIN {X 0,Y 608.442,Z 668.509,A -85,B 0,C 180,E1 -541.324,E2 -541.324} C_VEL
LIN {X 0,Y 608.421,Z 667.153,A -85,B 0,C 180,E1 -542.649,E2 -542.649} C_VEL
LIN {X 0,Y 608.428,Z 664.73,A -85,B 0,C 180,E1 -543.974,E2 -543.974} C_VEL
LIN {X 0,Y 608.436,Z 661.385,A -85,B 0,C 180,E1 -545.302,E2 -545.302} C_VEL
LIN {X 0,Y 608.439,Z 655.644,A -85,B 0,C 180,E1 -546.967,E2 -546.967} C_VEL
LIN {X 0,Y 608.453,Z 649.702,A -85,B 0,C 180,E1 -548.302,E2 -548.302} C_VEL
LIN {X 0,Y 608.437,Z 644.768,A -85,B 0,C 180,E1 -549.252,E2 -549.252} C_VEL
LIN {X 0,Y 607.775,Z 642.058,A -85,B 0,C 180,E1 -549.743,E2 -549.743} C_VEL
LIN {X 0,Y 602.067,Z 632.593,A -85,B 0,C 180,E1 -551.302,E2 -551.302} C_VEL
LIN {X 0,Y 601.443,Z 629.279,A -85,B 0,C 180,E1 -551.769,E2 -551.769} C_VEL
LIN {X 0,Y 601.473,Z 619.324,A -85,B 0,C 180,E1 -552.999,E2 -552.999} C_VEL
LIN {X 0,Y 601.54,Z 607.972,A -85,B 0,C 180,E1 -554.203,E2 -554.203} C_VEL
LIN {X 0,Y 601.6,Z 595.578,A -85,B 0,C 180,E1 -555.326,E2 -555.326} C_VEL
LIN {X 0,Y 601.696,Z 582.147,A -85,B 0,C 180,E1 -556.364,E2 -556.364} C_VEL
LIN {X 0,Y 601.805,Z 567.319,A -85,B 0,C 180,E1 -557.325,E2 -557.325} C_VEL
LIN {X 0,Y 601.861,Z 552.657,A -85,B 0,C 180,E1 -558.114,E2 -558.114} C_VEL
LIN {X 0,Y 601.95,Z 537.018,A -85,B 0,C 180,E1 -558.803,E2 -558.803} C_VEL
LIN {X 0,Y 602.029,Z 519.966,A -85,B 0,C 180,E1 -559.389,E2 -559.389} C_VEL
LIN {X 0,Y 602.101,Z 503.531,A -85,B 0,C 180,E1 -559.808,E2 -559.808} C_VEL
LIN {X 0,Y 601.96,Z 486.063,A -85,B 0,C 180,E1 -560.106,E2 -560.106} C_VEL
LIN {X 0,Y 601.384,Z 483.89,A -85,B 0,C 180,E1 -560.167,E2 -560.167} C_VEL
LIN {X 0,Y 601.415,Z 483.883,A -85,B 0,C 180,E1 -562.683,E2 -562.683} C_VEL
LIN {X 0,Y 601.4,Z 483.886,A -85,B 0,C 180,E1 -564.879,E2 -564.879} C_VEL
LIN {X 0,Y 601.415,Z 483.886,A -85,B 0,C 180,E1 -567.362,E2 -567.362} C_VEL
LIN {X 0,Y 601.432,Z 483.883,A -85,B 0,C 180,E1 -570.164,E2 -570.164} C_VEL
LIN {X 0,Y 601.423,Z 483.882,A -85,B 0,C 180,E1 -572.715,E2 -572.715} C_VEL
LIN {X 0,Y 601.404,Z 483.884,A -85,B 0,C 180,E1 -575.113,E2 -575.113} C_VEL
LIN {X 0,Y 601.437,Z 483.884,A -85,B 0,C 180,E1 -577.419,E2 -577.419} C_VEL
LIN {X 0,Y 601.416,Z 483.883,A -85,B 0,C 180,E1 -579.995,E2 -579.995} C_VEL
LIN {X 0,Y 601.412,Z 483.883,A -85,B 0,C 180,E1 -582.671,E2 -582.671} C_VEL
LIN {X 0,Y 601.431,Z 483.88,A -85,B 0,C 180,E1 -585.482,E2 -585.482} C_VEL
LIN {X 0,Y 601.427,Z 483.881,A -85,B 0,C 180,E1 -588.407,E2 -588.407} C_VEL
LIN {X 0,Y 601.433,Z 483.88,A -85,B 0,C 180,E1 -590.875,E2 -590.875} C_VEL
LIN {X 0,Y 601.407,Z 483.886,A -85,B 0,C 180,E1 -593.417,E2 -593.417} C_VEL
LIN {X 0,Y 601.437,Z 483.885,A -85,B 0,C 180,E1 -596.064,E2 -596.064} C_VEL
LIN {X 0,Y 601.425,Z 483.882,A -85,B 0,C 180,E1 -598.545,E2 -598.545} C_VEL
LIN {X 0,Y 601.429,Z 483.881,A -85,B 0,C 180,E1 -601.373,E2 -601.373} C_VEL
LIN {X 0,Y 601.407,Z 483.884,A -85,B 0,C 180,E1 -603.636,E2 -603.636} C_VEL
LIN {X 0,Y 601.433,Z 483.977,A -85,B 0,C 180,E1 -605.95,E2 -605.95} C_VEL
LIN {X 0,Y 601.422,Z 488.063,A -85,B 0,C 180,E1 -608.041,E2 -608.041} C_VEL
LIN {X 0,Y 601.422,Z 493.358,A -85,B 0,C 180,E1 -610.901,E2 -610.901} C_VEL
LIN {X 0,Y 601.396,Z 498.742,A -85,B 0,C 180,E1 -613.711,E2 -613.711} C_VEL
LIN {X 0,Y 601.418,Z 504.208,A -85,B 0,C 180,E1 -616.484,E2 -616.484} C_VEL
LIN {X 0,Y 601.383,Z 509.757,A -85,B 0,C 180,E1 -619.223,E2 -619.223} C_VEL
LIN {X 0,Y 601.389,Z 515.381,A -85,B 0,C 180,E1 -621.938,E2 -621.938} C_VEL
LIN {X 0,Y 601.385,Z 521.666,A -85,B 0,C 180,E1 -624.908,E2 -624.908} C_VEL
LIN {X 0,Y 602.131,Z 525.049,A -85,B 0,C 180,E1 -624.977,E2 -624.977} C_VEL
LIN {X 0,Y 602.131,Z 541.841,A -85,B 0,C 180,E1 -625.25,E2 -625.25} C_VEL
LIN {X 0,Y 602.045,Z 558.112,A -85,B 0,C 180,E1 -625.648,E2 -625.648} C_VEL
LIN {X 0,Y 601.953,Z 573.529,A -85,B 0,C 180,E1 -626.15,E2 -626.15} C_VEL
LIN {X 0,Y 601.883,Z 589.469,A -85,B 0,C 180,E1 -626.82,E2 -626.82} C_VEL
LIN {X 0,Y 601.817,Z 605.446,A -85,B 0,C 180,E1 -627.657,E2 -627.657} C_VEL
LIN {X 0,Y 601.713,Z 619.957,A -85,B 0,C 180,E1 -628.577,E2 -628.577} C_VEL
LIN {X 0,Y 601.629,Z 633.34,A -85,B 0,C 180,E1 -629.581,E2 -629.581} C_VEL
LIN {X 0,Y 601.56,Z 645.708,A -85,B 0,C 180,E1 -630.669,E2 -630.669} C_VEL
LIN {X 0,Y 601.49,Z 657.146,A -85,B 0,C 180,E1 -631.841,E2 -631.841} C_VEL
LIN {X 0,Y 601.448,Z 668.253,A -85,B 0,C 180,E1 -633.181,E2 -633.181} C_VEL
LIN {X 0,Y 601.407,Z 677.611,A -85,B 0,C 180,E1 -634.523,E2 -634.523} C_VEL
LIN {X 0,Y 601.384,Z 684.609,A -85,B 0,C 180,E1 -635.7,E2 -635.7} C_VEL
LIN {X 0,Y 601.37,Z 691.415,A -85,B 0,C 180,E1 -637.048,E2 -637.048} C_VEL
LIN {X 0,Y 601.358,Z 696.959,A -85,B 0,C 180,E1 -638.399,E2 -638.399} C_VEL
LIN {X 0,Y 601.336,Z 700.414,A -85,B 0,C 180,E1 -639.416,E2 -639.416} C_VEL
LIN {X 0,Y 601.334,Z 704.509,A -85,B 0,C 180,E1 -640.965,E2 -640.965} C_VEL
LIN {X 0,Y 601.337,Z 706.717,A -85,B 0,C 180,E1 -642.143,E2 -642.143} C_VEL
LIN {X 0,Y 601.333,Z 708.348,A -85,B 0,C 180,E1 -643.517,E2 -643.517} C_VEL
LIN {X 0,Y 601.307,Z 708.972,A -85,B 0,C 180,E1 -644.899,E2 -644.899} C_VEL
LIN {X 0,Y 601.318,Z 708.339,A -85,B 0,C 180,E1 -646.586,E2 -646.586} C_VEL
LIN {X 0,Y 601.309,Z 707.137,A -85,B 0,C 180,E1 -647.69,E2 -647.69} C_VEL
LIN {X 0,Y 601.312,Z 704.559,A -85,B 0,C 180,E1 -649.101,E2 -649.101} C_VEL
LIN {X 0,Y 601.364,Z 700.077,A -85,B 0,C 180,E1 -650.78,E2 -650.78} C_VEL
LIN {X 0,Y 601.346,Z 694.696,A -85,B 0,C 180,E1 -652.279,E2 -652.279} C_VEL
LIN {X 0,Y 601.369,Z 687.89,A -85,B 0,C 180,E1 -653.777,E2 -653.777} C_VEL
LIN {X 0,Y 601.381,Z 679.621,A -85,B 0,C 180,E1 -655.248,E2 -655.248} C_VEL
LIN {X 0,Y 601.421,Z 670.88,A -85,B 0,C 180,E1 -656.549,E2 -656.549} C_VEL
LIN {X 0,Y 601.458,Z 660.496,A -85,B 0,C 180,E1 -657.864,E2 -657.864} C_VEL
LIN {X 0,Y 601.518,Z 649.471,A -85,B 0,C 180,E1 -659.057,E2 -659.057} C_VEL
LIN {X 0,Y 601.614,Z 637.35,A -85,B 0,C 180,E1 -660.178,E2 -660.178} C_VEL
LIN {X 0,Y 601.691,Z 623.566,A -85,B 0,C 180,E1 -661.262,E2 -661.262} C_VEL
LIN {X 0,Y 601.771,Z 609.424,A -85,B 0,C 180,E1 -662.197,E2 -662.197} C_VEL
LIN {X 0,Y 601.859,Z 595.943,A -85,B 0,C 180,E1 -662.948,E2 -662.948} C_VEL
LIN {X 0,Y 601.948,Z 581.328,A -85,B 0,C 180,E1 -663.63,E2 -663.63} C_VEL
LIN {X 0,Y 601.992,Z 565.103,A -85,B 0,C 180,E1 -664.232,E2 -664.232} C_VEL
LIN {X 0,Y 602.095,Z 548.494,A -85,B 0,C 180,E1 -664.694,E2 -664.694} C_VEL
LIN {X 0,Y 602.126,Z 532.97,A -85,B 0,C 180,E1 -665,E2 -665} C_VEL
LIN {X 0,Y 602.029,Z 524.398,A -85,B 0,C 180,E1 -665.124,E2 -665.124} C_VEL
LIN {X 0,Y 601.347,Z 521.633,A -85,B 0,C 180,E1 -665.199,E2 -665.199} C_VEL
LIN {X 0,Y 601.357,Z 516.914,A -85,B 0,C 180,E1 -667.423,E2 -667.423} C_VEL
LIN {X 0,Y 601.363,Z 511.547,A -85,B 0,C 180,E1 -669.997,E2 -669.997} C_VEL
LIN {X 0,Y 601.378,Z 506.089,A -85,B 0,C 180,E1 -672.672,E2 -672.672} C_VEL
LIN {X 0,Y 601.392,Z 500.502,A -85,B 0,C 180,E1 -675.478,E2 -675.478} C_VEL
LIN {X 0,Y 601.422,Z 494.842,A -85,B 0,C 180,E1 -678.405,E2 -678.405} C_VEL
LIN {X 0,Y 601.431,Z 490.214,A -85,B 0,C 180,E1 -680.875,E2 -680.875} C_VEL
LIN {X 0,Y 601.41,Z 485.476,A -85,B 0,C 180,E1 -683.417,E2 -683.417} C_VEL
LIN {X 0,Y 601.445,Z 483.881,A -85,B 0,C 180,E1 -684.249,E2 -684.249} C_VEL
LIN {X 0,Y 601.428,Z 483.886,A -85,B 0,C 180,E1 -686.686,E2 -686.686} C_VEL
LIN {X 0,Y 601.424,Z 483.883,A -85,B 0,C 180,E1 -689.058,E2 -689.058} C_VEL
LIN {X 0,Y 601.43,Z 483.881,A -85,B 0,C 180,E1 -691.373,E2 -691.373} C_VEL
LIN {X 0,Y 601.418,Z 483.882,A -85,B 0,C 180,E1 -694.129,E2 -694.129} C_VEL
LIN {X 0,Y 601.418,Z 483.883,A -85,B 0,C 180,E1 -696.589,E2 -696.589} C_VEL
LIN {X 0,Y 601.427,Z 483.881,A -85,B 0,C 180,E1 -699.478,E2 -699.478} C_VEL
LIN {X 0,Y 601.4,Z 483.884,A -85,B 0,C 180,E1 -702.311,E2 -702.311} C_VEL
LIN {X 0,Y 601.427,Z 483.881,A -85,B 0,C 180,E1 -705.103,E2 -705.103} C_VEL
LIN {X 0,Y 601.415,Z 483.882,A -85,B 0,C 180,E1 -707.857,E2 -707.857} C_VEL
LIN {X 0,Y 601.418,Z 483.882,A -85,B 0,C 180,E1 -710.584,E2 -710.584} C_VEL
LIN {X 0,Y 601.445,Z 483.879,A -85,B 0,C 180,E1 -713.322,E2 -713.322} C_VEL
LIN {X 0,Y 601.399,Z 483.884,A -85,B 0,C 180,E1 -715.979,E2 -715.979} C_VEL
LIN {X 0,Y 601.425,Z 483.881,A -85,B 0,C 180,E1 -718.661,E2 -718.661} C_VEL
LIN {X 0,Y 601.423,Z 483.881,A -85,B 0,C 180,E1 -721.339,E2 -721.339} C_VEL
LIN {X 0,Y 601.4,Z 483.884,A -85,B 0,C 180,E1 -724.02,E2 -724.02} C_VEL
LIN {X 0,Y 601.441,Z 483.879,A -85,B 0,C 180,E1 -726.71,E2 -726.71} C_VEL
LIN {X 0,Y 601.411,Z 483.883,A -85,B 0,C 180,E1 -729.416,E2 -729.416} C_VEL
LIN {X 0,Y 601.414,Z 483.882,A -85,B 0,C 180,E1 -732.142,E2 -732.142} C_VEL
LIN {X 0,Y 601.427,Z 483.881,A -85,B 0,C 180,E1 -734.897,E2 -734.897} C_VEL
LIN {X 0,Y 601.427,Z 483.884,A -85,B 0,C 180,E1 -736.986,E2 -736.986} C_VEL
LIN {X 0,Y 601.402,Z 483.888,A -85,B 0,C 180,E1 -739.809,E2 -739.809} C_VEL
LIN {X 0,Y 601.446,Z 483.88,A -85,B 0,C 180,E1 -742.681,E2 -742.681} C_VEL
LIN {X 0,Y 601.404,Z 483.884,A -85,B 0,C 180,E1 -744.878,E2 -744.878} C_VEL
LIN {X 0,Y 601.418,Z 483.887,A -85,B 0,C 180,E1 -747.867,E2 -747.867} C_VEL
LIN {X 0,Y 601.438,Z 483.88,A -85,B 0,C 180,E1 -750.163,E2 -750.163} C_VEL
LIN {X 0,Y 601.422,Z 483.882,A -85,B 0,C 180,E1 -752.718,E2 -752.718} C_VEL
LIN {X 0,Y 601.414,Z 483.883,A -85,B 0,C 180,E1 -755.117,E2 -755.117} C_VEL
LIN {X 0,Y 601.428,Z 483.885,A -85,B 0,C 180,E1 -757.419,E2 -757.419} C_VEL
LIN {X 0,Y 601.414,Z 483.887,A -85,B 0,C 180,E1 -759.995,E2 -759.995} C_VEL
LIN {X 0,Y 601.403,Z 483.887,A -85,B 0,C 180,E1 -762.671,E2 -762.671} C_VEL
LIN {X 0,Y 601.416,Z 483.887,A -85,B 0,C 180,E1 -765.483,E2 -765.483} C_VEL
LIN {X 0,Y 601.425,Z 483.884,A -85,B 0,C 180,E1 -768.406,E2 -768.406} C_VEL
LIN {X 0,Y 601.439,Z 483.995,A -85,B 0,C 180,E1 -769.85,E2 -769.85} C_VEL
LIN {X 0,Y 601.919,Z 487.24,A -85,B 0,C 180,E1 -770.665,E2 -770.665} C_VEL
LIN {X 0,Y 601.857,Z 499.184,A -85,B 0,C 180,E1 -773.451,E2 -773.451} C_VEL
LIN {X 0,Y 601.792,Z 512.141,A -85,B 0,C 180,E1 -776.363,E2 -776.363} C_VEL
LIN {X 0,Y 601.683,Z 524.612,A -85,B 0,C 180,E1 -779.074,E2 -779.074} C_VEL
LIN {X 0,Y 601.648,Z 537.326,A -85,B 0,C 180,E1 -781.766,E2 -781.766} C_VEL
LIN {X 0,Y 601.59,Z 550.04,A -85,B 0,C 180,E1 -784.391,E2 -784.391} C_VEL
LIN {X 0,Y 601.54,Z 562.754,A -85,B 0,C 180,E1 -786.96,E2 -786.96} C_VEL
LIN {X 0,Y 601.508,Z 577.142,A -85,B 0,C 180,E1 -789.811,E2 -789.811} C_VEL
LIN {X 0,Y 602.121,Z 581.082,A -85,B 0,C 180,E1 -789.883,E2 -789.883} C_VEL
LIN {X 0,Y 602.089,Z 600.112,A -85,B 0,C 180,E1 -790.171,E2 -790.171} C_VEL
LIN {X 0,Y 602.051,Z 616.961,A -85,B 0,C 180,E1 -790.569,E2 -790.569} C_VEL
LIN {X 0,Y 601.99,Z 632.39,A -85,B 0,C 180,E1 -791.063,E2 -791.063} C_VEL
LIN {X 0,Y 601.881,Z 648.06,A -85,B 0,C 180,E1 -791.712,E2 -791.712} C_VEL
LIN {X 0,Y 601.802,Z 661.892,A -85,B 0,C 180,E1 -792.413,E2 -792.413} C_VEL
LIN {X 0,Y 601.723,Z 676.317,A -85,B 0,C 180,E1 -793.283,E2 -793.283} C_VEL
LIN {X 0,Y 601.66,Z 689.703,A -85,B 0,C 180,E1 -794.242,E2 -794.242} C_VEL
LIN {X 0,Y 601.583,Z 702.017,A -85,B 0,C 180,E1 -795.281,E2 -795.281} C_VEL
LIN {X 0,Y 601.489,Z 714.27,A -85,B 0,C 180,E1 -796.487,E2 -796.487} C_VEL
LIN {X 0,Y 601.451,Z 724.698,A -85,B 0,C 180,E1 -797.688,E2 -797.688} C_VEL
LIN {X 0,Y 601.428,Z 734.359,A -85,B 0,C 180,E1 -798.986,E2 -798.986} C_VEL
LIN {X 0,Y 601.388,Z 742.289,A -85,B 0,C 180,E1 -800.245,E2 -800.245} C_VEL
LIN {X 0,Y 601.364,Z 749.49,A -85,B 0,C 180,E1 -801.601,E2 -801.601} C_VEL
LIN {X 0,Y 601.367,Z 755.472,A -85,B 0,C 180,E1 -802.952,E2 -802.952} C_VEL
LIN {X 0,Y 601.347,Z 761.248,A -85,B 0,C 180,E1 -804.636,E2 -804.636} C_VEL
LIN {X 0,Y 601.34,Z 764.634,A -85,B 0,C 180,E1 -805.98,E2 -805.98} C_VEL
LIN {X 0,Y 601.312,Z 767.087,A -85,B 0,C 180,E1 -807.321,E2 -807.321} C_VEL
LIN {X 0,Y 601.345,Z 768.478,A -85,B 0,C 180,E1 -808.661,E2 -808.661} C_VEL
LIN {X 0,Y 601.33,Z 769,A -85,B 0,C 180,E1 -810.001,E2 -810.001} C_VEL
LIN {X 0,Y 601.345,Z 768.477,A -85,B 0,C 180,E1 -811.34,E2 -811.34} C_VEL
LIN {X 0,Y 601.312,Z 767.085,A -85,B 0,C 180,E1 -812.68,E2 -812.68} C_VEL
LIN {X 0,Y 601.34,Z 764.631,A -85,B 0,C 180,E1 -814.022,E2 -814.022} C_VEL
LIN {X 0,Y 601.347,Z 761.243,A -85,B 0,C 180,E1 -815.365,E2 -815.365} C_VEL
LIN {X 0,Y 601.368,Z 755.466,A -85,B 0,C 180,E1 -817.049,E2 -817.049} C_VEL
LIN {X 0,Y 601.377,Z 747.854,A -85,B 0,C 180,E1 -818.739,E2 -818.739} C_VEL
LIN {X 0,Y 601.409,Z 739.242,A -85,B 0,C 180,E1 -820.266,E2 -820.266} C_VEL
LIN {X 0,Y 601.426,Z 729.964,A -85,B 0,C 180,E1 -821.63,E2 -821.63} C_VEL
LIN {X 0,Y 601.48,Z 720.417,A -85,B 0,C 180,E1 -822.827,E2 -822.827} C_VEL
LIN {X 0,Y 601.545,Z 709.616,A -85,B 0,C 180,E1 -823.997,E2 -823.997} C_VEL
LIN {X 0,Y 601.608,Z 697.136,A -85,B 0,C 180,E1 -825.153,E2 -825.153} C_VEL
LIN {X 0,Y 601.717,Z 682.702,A -85,B 0,C 180,E1 -826.28,E2 -826.28} C_VEL
LIN {X 0,Y 601.777,Z 668.008,A -85,B 0,C 180,E1 -827.239,E2 -827.239} C_VEL
LIN {X 0,Y 601.855,Z 653.502,A -85,B 0,C 180,E1 -828.026,E2 -828.026} C_VEL
LIN {X 0,Y 601.929,Z 638.077,A -85,B 0,C 180,E1 -828.716,E2 -828.716} C_VEL
LIN {X 0,Y 602.056,Z 622.221,A -85,B 0,C 180,E1 -829.278,E2 -829.278} C_VEL
LIN {X 0,Y 602.08,Z 606.499,A -85,B 0,C 180,E1 -829.698,E2 -829.698} C_VEL
LIN {X 0,Y 602.131,Z 590.893,A -85,B 0,C 180,E1 -829.985,E2 -829.985} C_VEL
LIN {X 0,Y 601.944,Z 579.172,A -85,B 0,C 180,E1 -830.147,E2 -830.147} C_VEL
LIN {X 0,Y 601.499,Z 577.049,A -85,B 0,C 180,E1 -830.207,E2 -830.207} C_VEL
LIN {X 0,Y 601.541,Z 562.746,A -85,B 0,C 180,E1 -833.042,E2 -833.042} C_VEL
LIN {X 0,Y 601.59,Z 550.032,A -85,B 0,C 180,E1 -835.611,E2 -835.611} C_VEL
LIN {X 0,Y 601.65,Z 537.318,A -85,B 0,C 180,E1 -838.235,E2 -838.235} C_VEL
LIN {X 0,Y 601.684,Z 524.604,A -85,B 0,C 180,E1 -840.927,E2 -840.927} C_VEL
LIN {X 0,Y 601.793,Z 512.135,A -85,B 0,C 180,E1 -843.638,E2 -843.638} C_VEL
LIN {X 0,Y 601.862,Z 499.177,A -85,B 0,C 180,E1 -846.551,E2 -846.551} C_VEL
LIN {X 0,Y 601.929,Z 487.238,A -85,B 0,C 180,E1 -849.334,E2 -849.334} C_VEL
LIN {X 0,Y 601.411,Z 483.885,A -85,B 0,C 180,E1 -850.206,E2 -850.206} C_VEL
LIN {X 0,Y 601.417,Z 483.884,A -85,B 0,C 180,E1 -852.67,E2 -852.67} C_VEL
LIN {X 0,Y 601.427,Z 483.877,A -85,B 0,C 180,E1 -855.482,E2 -855.482} C_VEL
LIN {X 0,Y 601.425,Z 483.882,A -85,B 0,C 180,E1 -858.407,E2 -858.407} C_VEL
LIN {X 0,Y 601.437,Z 483.88,A -85,B 0,C 180,E1 -860.876,E2 -860.876} C_VEL
LIN {X 0,Y 601.402,Z 483.879,A -85,B 0,C 180,E1 -863.417,E2 -863.417} C_VEL
LIN {X 0,Y 601.433,Z 483.881,A -85,B 0,C 180,E1 -866.065,E2 -866.065} C_VEL
LIN {X 0,Y 601.42,Z 483.882,A -85,B 0,C 180,E1 -868.546,E2 -868.546} C_VEL
LIN {X 0,Y 601.434,Z 483.876,A -85,B 0,C 180,E1 -871.374,E2 -871.374} C_VEL
LIN {X 0,Y 601.416,Z 483.885,A -85,B 0,C 180,E1 -874.132,E2 -874.132} C_VEL
LIN {X 0,Y 601.421,Z 483.878,A -85,B 0,C 180,E1 -876.59,E2 -876.59} C_VEL
LIN {X 0,Y 601.423,Z 483.882,A -85,B 0,C 180,E1 -879.478,E2 -879.478} C_VEL
LIN {X 0,Y 601.379,Z 483.891,A -85,B 0,C 180,E1 -879.923,E2 -879.923} C_VEL
LIN {X 0,Y 602.158,Z 487.156,A -85,B 0,C 180,E1 -880.006,E2 -880.006} C_VEL
LIN {X 0,Y 602.106,Z 503.507,A -85,B 0,C 180,E1 -880.282,E2 -880.282} C_VEL
LIN {X 0,Y 602.051,Z 519.209,A -85,B 0,C 180,E1 -880.679,E2 -880.679} C_VEL
LIN {X 0,Y 601.971,Z 534.732,A -85,B 0,C 180,E1 -881.198,E2 -881.198} C_VEL
LIN {X 0,Y 601.894,Z 549.015,A -85,B 0,C 180,E1 -881.8,E2 -881.8} C_VEL
LIN {X 0,Y 601.796,Z 564.215,A -85,B 0,C 180,E1 -882.587,E2 -882.587} C_VEL
LIN {X 0,Y 601.714,Z 577.852,A -85,B 0,C 180,E1 -883.433,E2 -883.433} C_VEL
LIN {X 0,Y 601.637,Z 591.311,A -85,B 0,C 180,E1 -884.415,E2 -884.415} C_VEL
LIN {X 0,Y 601.565,Z 603.446,A -85,B 0,C 180,E1 -885.453,E2 -885.453} C_VEL
LIN {X 0,Y 601.497,Z 615.471,A -85,B 0,C 180,E1 -886.658,E2 -886.658} C_VEL
LIN {X 0,Y 601.438,Z 625.702,A -85,B 0,C 180,E1 -887.858,E2 -887.858} C_VEL
LIN {X 0,Y 601.405,Z 635.636,A -85,B 0,C 180,E1 -889.224,E2 -889.224} C_VEL
LIN {X 0,Y 601.369,Z 643.993,A -85,B 0,C 180,E1 -890.584,E2 -890.584} C_VEL
LIN {X 0,Y 601.361,Z 650.893,A -85,B 0,C 180,E1 -891.938,E2 -891.938} C_VEL
LIN {X 0,Y 601.352,Z 657.004,A -85,B 0,C 180,E1 -893.411,E2 -893.411} C_VEL
LIN {X 0,Y 601.35,Z 661.108,A -85,B 0,C 180,E1 -894.636,E2 -894.636} C_VEL
LIN {X 0,Y 601.337,Z 664.538,A -85,B 0,C 180,E1 -895.979,E2 -895.979} C_VEL
LIN {X 0,Y 601.322,Z 667.015,A -85,B 0,C 180,E1 -897.321,E2 -897.321} C_VEL
LIN {X 0,Y 601.341,Z 668.448,A -85,B 0,C 180,E1 -898.661,E2 -898.661} C_VEL
LIN {X 0,Y 601.332,Z 668.996,A -85,B 0,C 180,E1 -900,E2 -900} C_VEL
LIN {X 0,Y 601.342,Z 668.511,A -85,B 0,C 180,E1 -901.34,E2 -901.34} C_VEL
LIN {X 0,Y 601.32,Z 667.15,A -85,B 0,C 180,E1 -902.68,E2 -902.68} C_VEL
LIN {X 0,Y 601.338,Z 664.73,A -85,B 0,C 180,E1 -904.021,E2 -904.021} C_VEL
LIN {X 0,Y 601.348,Z 661.382,A -85,B 0,C 180,E1 -905.365,E2 -905.365} C_VEL
LIN {X 0,Y 601.367,Z 655.64,A -85,B 0,C 180,E1 -907.049,E2 -907.049} C_VEL
LIN {X 0,Y 601.391,Z 648.081,A -85,B 0,C 180,E1 -908.739,E2 -908.739} C_VEL
LIN {X 0,Y 601.409,Z 639.516,A -85,B 0,C 180,E1 -910.266,E2 -910.266} C_VEL
LIN {X 0,Y 601.43,Z 630.294,A -85,B 0,C 180,E1 -911.629,E2 -911.629} C_VEL
LIN {X 0,Y 601.443,Z 629.279,A -85,B 0,C 180,E1 -911.769,E2 -911.769} C_VEL
LIN {X 0,Y 600.814,Z 625.935,A -85,B 0,C 180,E1 -912.23,E2 -912.23} C_VEL
LIN {X 0,Y 597.976,Z 620.421,A -85,B 0,C 180,E1 -912.971,E2 -912.971} C_VEL
LIN {X 0,Y 595.148,Z 614.53,A -85,B 0,C 180,E1 -913.69,E2 -913.69} C_VEL
LIN {X 0,Y 594.537,Z 610.597,A -85,B 0,C 180,E1 -914.112,E2 -914.112} C_VEL
LIN {X 0,Y 594.644,Z 598.631,A -85,B 0,C 180,E1 -915.247,E2 -915.247} C_VEL
LIN {X 0,Y 594.8,Z 585.639,A -85,B 0,C 180,E1 -916.298,E2 -916.298} C_VEL
LIN {X 0,Y 594.897,Z 571.565,A -85,B 0,C 180,E1 -917.267,E2 -917.267} C_VEL
LIN {X 0,Y 595.041,Z 557.894,A -85,B 0,C 180,E1 -918.062,E2 -918.062} C_VEL
LIN {X 0,Y 595.162,Z 542.302,A -85,B 0,C 180,E1 -918.809,E2 -918.809} C_VEL
LIN {X 0,Y 595.256,Z 526.934,A -85,B 0,C 180,E1 -919.394,E2 -919.394} C_VEL
LIN {X 0,Y 595.37,Z 510.196,A -85,B 0,C 180,E1 -919.884,E2 -919.884} C_VEL
LIN {X 0,Y 595.467,Z 493.877,A -85,B 0,C 180,E1 -920.218,E2 -920.218} C_VEL
LIN {X 0,Y 595.278,Z 487.624,A -85,B 0,C 180,E1 -920.319,E2 -920.319} C_VEL
LIN {X 0,Y 594.366,Z 484.765,A -85,B 0,C 180,E1 -920.393,E2 -920.393} C_VEL
LIN {X 0,Y 594.367,Z 484.763,A -85,B 0,C 180,E1 -922.968,E2 -922.968} C_VEL
LIN {X 0,Y 594.378,Z 484.759,A -85,B 0,C 180,E1 -925.193,E2 -925.193} C_VEL
LIN {X 0,Y 594.371,Z 484.764,A -85,B 0,C 180,E1 -927.524,E2 -927.524} C_VEL
LIN {X 0,Y 594.389,Z 484.762,A -85,B 0,C 180,E1 -930.328,E2 -930.328} C_VEL
LIN {X 0,Y 594.382,Z 484.761,A -85,B 0,C 180,E1 -932.95,E2 -932.95} C_VEL
LIN {X 0,Y 594.362,Z 484.76,A -85,B 0,C 180,E1 -935.409,E2 -935.409} C_VEL
LIN {X 0,Y 594.385,Z 484.758,A -85,B 0,C 180,E1 -937.941,E2 -937.941} C_VEL
LIN {X 0,Y 594.377,Z 484.759,A -85,B 0,C 180,E1 -940.822,E2 -940.822} C_VEL
LIN {X 0,Y 594.371,Z 484.763,A -85,B 0,C 180,E1 -943.3,E2 -943.3} C_VEL
LIN {X 0,Y 594.388,Z 484.761,A -85,B 0,C 180,E1 -946.159,E2 -946.159} C_VEL
LIN {X 0,Y 594.382,Z 484.76,A -85,B 0,C 180,E1 -949.178,E2 -949.178} C_VEL
LIN {X 0,Y 594.388,Z 484.759,A -85,B 0,C 180,E1 -952.059,E2 -952.059} C_VEL
LIN {X 0,Y 594.355,Z 484.766,A -85,B 0,C 180,E1 -954.677,E2 -954.677} C_VEL
LIN {X 0,Y 594.384,Z 484.759,A -85,B 0,C 180,E1 -957.088,E2 -957.088} C_VEL
LIN {X 0,Y 594.392,Z 484.757,A -85,B 0,C 180,E1 -959.672,E2 -959.672} C_VEL
LIN {X 0,Y 594.381,Z 484.758,A -85,B 0,C 180,E1 -962.539,E2 -962.539} C_VEL
LIN {X 0,Y 594.379,Z 484.762,A -85,B 0,C 180,E1 -964.807,E2 -964.807} C_VEL
LIN {X 0,Y 594.391,Z 484.93,A -85,B 0,C 180,E1 -966.018,E2 -966.018} C_VEL
LIN {X 0,Y 594.373,Z 489.796,A -85,B 0,C 180,E1 -968.496,E2 -968.496} C_VEL
LIN {X 0,Y 594.377,Z 495.114,A -85,B 0,C 180,E1 -971.382,E2 -971.382} C_VEL
LIN {X 0,Y 594.321,Z 500.515,A -85,B 0,C 180,E1 -974.217,E2 -974.217} C_VEL
LIN {X 0,Y 594.359,Z 504.616,A -85,B 0,C 180,E1 -976.32,E2 -976.32} C_VEL
LIN {X 0,Y 594.32,Z 510.161,A -85,B 0,C 180,E1 -979.093,E2 -979.093} C_VEL
LIN {X 0,Y 594.309,Z 515.784,A -85,B 0,C 180,E1 -981.841,E2 -981.841} C_VEL
LIN {X 0,Y 594.282,Z 521.664,A -85,B 0,C 180,E1 -984.656,E2 -984.656} C_VEL
LIN {X 0,Y 595.465,Z 527.276,A -85,B 0,C 180,E1 -984.772,E2 -984.772} C_VEL
LIN {X 0,Y 595.436,Z 544.351,A -85,B 0,C 180,E1 -985.069,E2 -985.069} C_VEL
LIN {X 0,Y 595.281,Z 560.602,A -85,B 0,C 180,E1 -985.492,E2 -985.492} C_VEL
LIN {X 0,Y 595.187,Z 576.967,A -85,B 0,C 180,E1 -986.064,E2 -986.064} C_VEL
LIN {X 0,Y 595.083,Z 593.039,A -85,B 0,C 180,E1 -986.783,E2 -986.783} C_VEL
LIN {X 0,Y 594.956,Z 607.061,A -85,B 0,C 180,E1 -987.545,E2 -987.545} C_VEL
LIN {X 0,Y 594.834,Z 621.329,A -85,B 0,C 180,E1 -988.476,E2 -988.476} C_VEL
LIN {X 0,Y 594.689,Z 635.518,A -85,B 0,C 180,E1 -989.576,E2 -989.576} C_VEL
LIN {X 0,Y 594.583,Z 647.537,A -85,B 0,C 180,E1 -990.677,E2 -990.677} C_VEL
LIN {X 0,Y 594.482,Z 658.696,A -85,B 0,C 180,E1 -991.862,E2 -991.862} C_VEL
LIN {X 0,Y 594.405,Z 669.558,A -85,B 0,C 180,E1 -993.219,E2 -993.219} C_VEL
LIN {X 0,Y 594.361,Z 678.759,A -85,B 0,C 180,E1 -994.577,E2 -994.577} C_VEL
LIN {X 0,Y 594.325,Z 687.362,A -85,B 0,C 180,E1 -996.109,E2 -996.109} C_VEL
LIN {X 0,Y 594.283,Z 693.652,A -85,B 0,C 180,E1 -997.474,E2 -997.474} C_VEL
LIN {X 0,Y 594.246,Z 698.839,A -85,B 0,C 180,E1 -998.843,E2 -998.843} C_VEL
LIN {X 0,Y 594.23,Z 702.857,A -85,B 0,C 180,E1 -1000.218,E2 -1000.218} C_VEL
LIN {X 0,Y 594.232,Z 705.884,A -85,B 0,C 180,E1 -1001.598,E2 -1001.598} C_VEL
LIN {X 0,Y 594.235,Z 707.861,A -85,B 0,C 180,E1 -1002.985,E2 -1002.985} C_VEL
LIN {X 0,Y 594.21,Z 708.853,A -85,B 0,C 180,E1 -1004.381,E2 -1004.381} C_VEL
LIN {X 0,Y 594.214,Z 708.836,A -85,B 0,C 180,E1 -1005.784,E2 -1005.784} C_VEL
LIN {X 0,Y 594.238,Z 707.755,A -85,B 0,C 180,E1 -1007.197,E2 -1007.197} C_VEL
LIN {X 0,Y 594.239,Z 705.116,A -85,B 0,C 180,E1 -1008.887,E2 -1008.887} C_VEL
LIN {X 0,Y 594.266,Z 701.408,A -85,B 0,C 180,E1 -1010.418,E2 -1010.418} C_VEL
LIN {X 0,Y 594.264,Z 696.594,A -85,B 0,C 180,E1 -1011.871,E2 -1011.871} C_VEL
LIN {X 0,Y 594.278,Z 690.473,A -85,B 0,C 180,E1 -1013.338,E2 -1013.338} C_VEL
LIN {X 0,Y 594.352,Z 682.865,A -85,B 0,C 180,E1 -1014.819,E2 -1014.819} C_VEL
LIN {X 0,Y 594.37,Z 674.84,A -85,B 0,C 180,E1 -1016.119,E2 -1016.119} C_VEL
LIN {X 0,Y 594.444,Z 665.071,A -85,B 0,C 180,E1 -1017.456,E2 -1017.456} C_VEL
LIN {X 0,Y 594.503,Z 653.578,A -85,B 0,C 180,E1 -1018.795,E2 -1018.795} C_VEL
LIN {X 0,Y 594.607,Z 641.996,A -85,B 0,C 180,E1 -1019.943,E2 -1019.943} C_VEL
LIN {X 0,Y 594.736,Z 629.165,A -85,B 0,C 180,E1 -1021.031,E2 -1021.031} C_VEL
LIN {X 0,Y 594.85,Z 615.028,A -85,B 0,C 180,E1 -1022.048,E2 -1022.048} C_VEL
LIN {X 0,Y 594.998,Z 600.67,A -85,B 0,C 180,E1 -1022.91,E2 -1022.91} C_VEL
LIN {X 0,Y 595.113,Z 585.683,A -85,B 0,C 180,E1 -1023.657,E2 -1023.657} C_VEL
LIN {X 0,Y 595.247,Z 570.806,A -85,B 0,C 180,E1 -1024.261,E2 -1024.261} C_VEL
LIN {X 0,Y 595.356,Z 554.214,A -85,B 0,C 180,E1 -1024.784,E2 -1024.784} C_VEL
LIN {X 0,Y 595.44,Z 536.185,A -85,B 0,C 180,E1 -1025.183,E2 -1025.183} C_VEL
LIN {X 0,Y 595.409,Z 526.158,A -85,B 0,C 180,E1 -1025.335,E2 -1025.335} C_VEL
LIN {X 0,Y 594.303,Z 521.638,A -85,B 0,C 180,E1 -1025.446,E2 -1025.446} C_VEL
LIN {X 0,Y 594.278,Z 516.411,A -85,B 0,C 180,E1 -1027.947,E2 -1027.947} C_VEL
LIN {X 0,Y 594.294,Z 510.538,A -85,B 0,C 180,E1 -1030.812,E2 -1030.812} C_VEL
LIN {X 0,Y 594.341,Z 505.547,A -85,B 0,C 180,E1 -1033.3,E2 -1033.3} C_VEL
LIN {X 0,Y 594.354,Z 499.957,A -85,B 0,C 180,E1 -1036.16,E2 -1036.16} C_VEL
LIN {X 0,Y 594.378,Z 495.437,A -85,B 0,C 180,E1 -1038.535,E2 -1038.535} C_VEL
LIN {X 0,Y 594.383,Z 490.346,A -85,B 0,C 180,E1 -1041.294,E2 -1041.294} C_VEL
LIN {X 0,Y 594.376,Z 485.094,A -85,B 0,C 180,E1 -1043.967,E2 -1043.967} C_VEL
LIN {X 0,Y 594.38,Z 484.762,A -85,B 0,C 180,E1 -1044.176,E2 -1044.176} C_VEL
LIN {X 0,Y 594.38,Z 484.76,A -85,B 0,C 180,E1 -1046.238,E2 -1046.238} C_VEL
LIN {X 0,Y 594.384,Z 484.759,A -85,B 0,C 180,E1 -1048.65,E2 -1048.65} C_VEL
LIN {X 0,Y 594.381,Z 484.761,A -85,B 0,C 180,E1 -1051.04,E2 -1051.04} C_VEL
LIN {X 0,Y 594.39,Z 484.758,A -85,B 0,C 180,E1 -1053.973,E2 -1053.973} C_VEL
LIN {X 0,Y 594.386,Z 484.762,A -85,B 0,C 180,E1 -1056.295,E2 -1056.295} C_VEL
LIN {X 0,Y 594.4,Z 484.758,A -85,B 0,C 180,E1 -1059.224,E2 -1059.224} C_VEL
LIN {X 0,Y 594.38,Z 484.76,A -85,B 0,C 180,E1 -1062.095,E2 -1062.095} C_VEL
LIN {X 0,Y 594.362,Z 484.764,A -85,B 0,C 180,E1 -1064.219,E2 -1064.219} C_VEL
LIN {X 0,Y 594.371,Z 484.763,A -85,B 0,C 180,E1 -1067.017,E2 -1067.017} C_VEL
LIN {X 0,Y 594.393,Z 484.761,A -85,B 0,C 180,E1 -1069.784,E2 -1069.784} C_VEL
LIN {X 0,Y 594.394,Z 484.761,A -85,B 0,C 180,E1 -1072.527,E2 -1072.527} C_VEL
LIN {X 0,Y 594.4,Z 484.761,A -85,B 0,C 180,E1 -1075.252,E2 -1075.252} C_VEL
LIN {X 0,Y 594.402,Z 484.76,A -85,B 0,C 180,E1 -1077.967,E2 -1077.967} C_VEL
LIN {X 0,Y 594.423,Z 484.758,A -85,B 0,C 180,E1 -1080.677,E2 -1080.677} C_VEL
LIN {X 0,Y 594.38,Z 484.763,A -85,B 0,C 180,E1 -1083.389,E2 -1083.389} C_VEL
LIN {X 0,Y 594.362,Z 484.765,A -85,B 0,C 180,E1 -1086.109,E2 -1086.109} C_VEL
LIN {X 0,Y 594.395,Z 484.761,A -85,B 0,C 180,E1 -1088.842,E2 -1088.842} C_VEL
LIN {X 0,Y 594.385,Z 484.762,A -85,B 0,C 180,E1 -1091.596,E2 -1091.596} C_VEL
LIN {X 0,Y 594.38,Z 484.762,A -85,B 0,C 180,E1 -1094.377,E2 -1094.377} C_VEL
LIN {X 0,Y 594.383,Z 484.758,A -85,B 0,C 180,E1 -1097.193,E2 -1097.193} C_VEL
LIN {X 0,Y 594.372,Z 484.761,A -85,B 0,C 180,E1 -1100.054,E2 -1100.054} C_VEL
LIN {X 0,Y 594.39,Z 484.757,A -85,B 0,C 180,E1 -1102.966,E2 -1102.966} C_VEL
LIN {X 0,Y 594.377,Z 484.762,A -85,B 0,C 180,E1 -1105.193,E2 -1105.193} C_VEL
LIN {X 0,Y 594.373,Z 484.761,A -85,B 0,C 180,E1 -1107.527,E2 -1107.527} C_VEL
LIN {X 0,Y 594.39,Z 484.76,A -85,B 0,C 180,E1 -1110.331,E2 -1110.331} C_VEL
LIN {X 0,Y 594.371,Z 484.761,A -85,B 0,C 180,E1 -1112.95,E2 -1112.95} C_VEL
LIN {X 0,Y 594.378,Z 484.759,A -85,B 0,C 180,E1 -1115.407,E2 -1115.407} C_VEL
LIN {X 0,Y 594.379,Z 484.759,A -85,B 0,C 180,E1 -1117.941,E2 -1117.941} C_VEL
LIN {X 0,Y 594.385,Z 484.758,A -85,B 0,C 180,E1 -1120.825,E2 -1120.825} C_VEL
LIN {X 0,Y 594.373,Z 484.761,A -85,B 0,C 180,E1 -1123.842,E2 -1123.842} C_VEL
LIN {X 0,Y 594.378,Z 484.763,A -85,B 0,C 180,E1 -1126.703,E2 -1126.703} C_VEL
LIN {X 0,Y 594.41,Z 484.856,A -85,B 0,C 180,E1 -1129.488,E2 -1129.488} C_VEL
LIN {X 0,Y 595.111,Z 488.287,A -85,B 0,C 180,E1 -1130.38,E2 -1130.38} C_VEL
LIN {X 0,Y 595.046,Z 499.184,A -85,B 0,C 180,E1 -1132.963,E2 -1132.963} C_VEL
LIN {X 0,Y 594.944,Z 511.51,A -85,B 0,C 180,E1 -1135.781,E2 -1135.781} C_VEL
LIN {X 0,Y 594.829,Z 524.612,A -85,B 0,C 180,E1 -1138.678,E2 -1138.678} C_VEL
LIN {X 0,Y 594.73,Z 537.326,A -85,B 0,C 180,E1 -1141.408,E2 -1141.408} C_VEL
LIN {X 0,Y 594.638,Z 549.354,A -85,B 0,C 180,E1 -1143.927,E2 -1143.927} C_VEL
LIN {X 0,Y 594.585,Z 562.754,A -85,B 0,C 180,E1 -1146.675,E2 -1146.675} C_VEL
LIN {X 0,Y 594.509,Z 577.114,A -85,B 0,C 180,E1 -1149.557,E2 -1149.557} C_VEL
LIN {X 0,Y 595.465,Z 581.814,A -85,B 0,C 180,E1 -1149.657,E2 -1149.657} C_VEL
LIN {X 0,Y 595.415,Z 600.112,A -85,B 0,C 180,E1 -1149.939,E2 -1149.939} C_VEL
LIN {X 0,Y 595.325,Z 616.962,A -85,B 0,C 180,E1 -1150.34,E2 -1150.34} C_VEL
LIN {X 0,Y 595.258,Z 632.778,A -85,B 0,C 180,E1 -1150.855,E2 -1150.855} C_VEL
LIN {X 0,Y 595.098,Z 648.062,A -85,B 0,C 180,E1 -1151.496,E2 -1151.496} C_VEL
LIN {X 0,Y 594.992,Z 663.459,A -85,B 0,C 180,E1 -1152.294,E2 -1152.294} C_VEL
LIN {X 0,Y 594.821,Z 678.563,A -85,B 0,C 180,E1 -1153.239,E2 -1153.239} C_VEL
LIN {X 0,Y 594.712,Z 691.863,A -85,B 0,C 180,E1 -1154.229,E2 -1154.229} C_VEL
LIN {X 0,Y 594.615,Z 703.95,A -85,B 0,C 180,E1 -1155.28,E2 -1155.28} C_VEL
LIN {X 0,Y 594.502,Z 715.898,A -85,B 0,C 180,E1 -1156.499,E2 -1156.499} C_VEL
LIN {X 0,Y 594.425,Z 726.06,A -85,B 0,C 180,E1 -1157.713,E2 -1157.713} C_VEL
LIN {X 0,Y 594.369,Z 735.935,A -85,B 0,C 180,E1 -1159.095,E2 -1159.095} C_VEL
LIN {X 0,Y 594.295,Z 744.233,A -85,B 0,C 180,E1 -1160.471,E2 -1160.471} C_VEL
LIN {X 0,Y 594.289,Z 751.108,A -85,B 0,C 180,E1 -1161.842,E2 -1161.842} C_VEL
LIN {X 0,Y 594.272,Z 756.72,A -85,B 0,C 180,E1 -1163.209,E2 -1163.209} C_VEL
LIN {X 0,Y 594.264,Z 761.248,A -85,B 0,C 180,E1 -1164.572,E2 -1164.572} C_VEL
LIN {X 0,Y 594.252,Z 764.635,A -85,B 0,C 180,E1 -1165.932,E2 -1165.932} C_VEL
LIN {X 0,Y 594.213,Z 767.088,A -85,B 0,C 180,E1 -1167.289,E2 -1167.289} C_VEL
LIN {X 0,Y 594.245,Z 768.478,A -85,B 0,C 180,E1 -1168.645,E2 -1168.645} C_VEL
LIN {X 0,Y 594.231,Z 769,A -85,B 0,C 180,E1 -1170.001,E2 -1170.001} C_VEL
LIN {X 0,Y 594.245,Z 768.477,A -85,B 0,C 180,E1 -1171.356,E2 -1171.356} C_VEL
LIN {X 0,Y 594.214,Z 767.085,A -85,B 0,C 180,E1 -1172.712,E2 -1172.712} C_VEL
LIN {X 0,Y 594.253,Z 764.632,A -85,B 0,C 180,E1 -1174.07,E2 -1174.07} C_VEL
LIN {X 0,Y 594.277,Z 760.183,A -85,B 0,C 180,E1 -1175.77,E2 -1175.77} C_VEL
LIN {X 0,Y 594.29,Z 755.466,A -85,B 0,C 180,E1 -1177.134,E2 -1177.134} C_VEL
LIN {X 0,Y 594.318,Z 747.854,A -85,B 0,C 180,E1 -1178.844,E2 -1178.844} C_VEL
LIN {X 0,Y 594.358,Z 739.242,A -85,B 0,C 180,E1 -1180.389,E2 -1180.389} C_VEL
LIN {X 0,Y 594.404,Z 729.964,A -85,B 0,C 180,E1 -1181.769,E2 -1181.769} C_VEL
LIN {X 0,Y 594.47,Z 720.417,A -85,B 0,C 180,E1 -1182.981,E2 -1182.981} C_VEL
LIN {X 0,Y 594.541,Z 708.943,A -85,B 0,C 180,E1 -1184.232,E2 -1184.232} C_VEL
LIN {X 0,Y 594.678,Z 697.136,A -85,B 0,C 180,E1 -1185.334,E2 -1185.334} C_VEL
LIN {X 0,Y 594.809,Z 683.879,A -85,B 0,C 180,E1 -1186.386,E2 -1186.386} C_VEL
LIN {X 0,Y 594.929,Z 669.421,A -85,B 0,C 180,E1 -1187.355,E2 -1187.355} C_VEL
LIN {X 0,Y 595.036,Z 655.251,A -85,B 0,C 180,E1 -1188.151,E2 -1188.151} C_VEL
LIN {X 0,Y 595.191,Z 640.198,A -85,B 0,C 180,E1 -1188.851,E2 -1188.851} C_VEL
LIN {X 0,Y 595.279,Z 624.332,A -85,B 0,C 180,E1 -1189.439,E2 -1189.439} C_VEL
LIN {X 0,Y 595.372,Z 608.326,A -85,B 0,C 180,E1 -1189.884,E2 -1189.884} C_VEL
LIN {X 0,Y 595.461,Z 592.399,A -85,B 0,C 180,E1 -1190.196,E2 -1190.196} C_VEL
LIN {X 0,Y 595.366,Z 580.837,A -85,B 0,C 180,E1 -1190.359,E2 -1190.359} C_VEL
LIN {X 0,Y 594.498,Z 577.049,A -85,B 0,C 180,E1 -1190.456,E2 -1190.456} C_VEL
LIN {X 0,Y 594.587,Z 562.746,A -85,B 0,C 180,E1 -1193.327,E2 -1193.327} C_VEL
LIN {X 0,Y 594.671,Z 548.097,A -85,B 0,C 180,E1 -1196.333,E2 -1196.333} C_VEL
LIN {X 0,Y 594.734,Z 535.318,A -85,B 0,C 180,E1 -1199.019,E2 -1199.019} C_VEL
LIN {X 0,Y 594.834,Z 522.816,A -85,B 0,C 180,E1 -1201.714,E2 -1201.714} C_VEL
LIN {X 0,Y 594.949,Z 510.074,A -85,B 0,C 180,E1 -1204.543,E2 -1204.543} C_VEL
LIN {X 0,Y 595.061,Z 497.776,A -85,B 0,C 180,E1 -1207.366,E2 -1207.366} C_VEL
LIN {X 0,Y 595.095,Z 488.279,A -85,B 0,C 180,E1 -1209.623,E2 -1209.623} C_VEL
LIN {X 0,Y 594.372,Z 484.764,A -85,B 0,C 180,E1 -1210.567,E2 -1210.567} C_VEL
LIN {X 0,Y 594.382,Z 484.758,A -85,B 0,C 180,E1 -1213.298,E2 -1213.298} C_VEL
LIN {X 0,Y 594.383,Z 484.755,A -85,B 0,C 180,E1 -1216.159,E2 -1216.159} C_VEL
LIN {X 0,Y 594.379,Z 484.756,A -85,B 0,C 180,E1 -1219.178,E2 -1219.178} C_VEL
LIN {X 0,Y 594.384,Z 484.757,A -85,B 0,C 180,E1 -1222.059,E2 -1222.059} C_VEL
LIN {X 0,Y 594.363,Z 484.762,A -85,B 0,C 180,E1 -1224.675,E2 -1224.675} C_VEL
LIN {X 0,Y 594.379,Z 484.755,A -85,B 0,C 180,E1 -1227.089,E2 -1227.089} C_VEL
LIN {X 0,Y 594.387,Z 484.756,A -85,B 0,C 180,E1 -1229.672,E2 -1229.672} C_VEL
LIN {X 0,Y 594.375,Z 484.758,A -85,B 0,C 180,E1 -1232.539,E2 -1232.539} C_VEL
LIN {X 0,Y 594.377,Z 484.755,A -85,B 0,C 180,E1 -1234.807,E2 -1234.807} C_VEL
LIN {X 0,Y 594.365,Z 484.758,A -85,B 0,C 180,E1 -1237.265,E2 -1237.265} C_VEL
LIN {X 0,Y 594.369,Z 484.765,A -85,B 0,C 180,E1 -1239.698,E2 -1239.698} C_VEL
LIN {X 0,Y 595.49,Z 488.748,A -85,B 0,C 180,E1 -1239.794,E2 -1239.794} C_VEL
LIN {X 0,Y 595.405,Z 505.639,A -85,B 0,C 180,E1 -1240.095,E2 -1240.095} C_VEL
LIN {X 0,Y 595.305,Z 521.514,A -85,B 0,C 180,E1 -1240.518,E2 -1240.518} C_VEL
LIN {X 0,Y 595.198,Z 537.832,A -85,B 0,C 180,E1 -1241.099,E2 -1241.099} C_VEL
LIN {X 0,Y 595.051,Z 552.653,A -85,B 0,C 180,E1 -1241.761,E2 -1241.761} C_VEL
LIN {X 0,Y 594.966,Z 567.306,A -85,B 0,C 180,E1 -1242.558,E2 -1242.558} C_VEL
LIN {X 0,Y 594.805,Z 582.085,A -85,B 0,C 180,E1 -1243.527,E2 -1243.527} C_VEL
LIN {X 0,Y 594.679,Z 595.561,A -85,B 0,C 180,E1 -1244.579,E2 -1244.579} C_VEL
LIN {X 0,Y 594.543,Z 608.492,A -85,B 0,C 180,E1 -1245.768,E2 -1245.768} C_VEL
LIN {X 0,Y 594.469,Z 620.047,A -85,B 0,C 180,E1 -1247.02,E2 -1247.02} C_VEL
LIN {X 0,Y 594.408,Z 630.892,A -85,B 0,C 180,E1 -1248.405,E2 -1248.405} C_VEL
LIN {X 0,Y 594.364,Z 640.002,A -85,B 0,C 180,E1 -1249.784,E2 -1249.784} C_VEL
LIN {X 0,Y 594.321,Z 647.626,A -85,B 0,C 180,E1 -1251.157,E2 -1251.157} C_VEL
LIN {X 0,Y 594.282,Z 653.865,A -85,B 0,C 180,E1 -1252.526,E2 -1252.526} C_VEL
LIN {X 0,Y 594.252,Z 658.991,A -85,B 0,C 180,E1 -1253.89,E2 -1253.89} C_VEL
LIN {X 0,Y 594.23,Z 662.944,A -85,B 0,C 180,E1 -1255.251,E2 -1255.251} C_VEL
LIN {X 0,Y 594.253,Z 665.914,A -85,B 0,C 180,E1 -1256.61,E2 -1256.61} C_VEL
LIN {X 0,Y 594.23,Z 667.843,A -85,B 0,C 180,E1 -1257.967,E2 -1257.967} C_VEL
LIN {X 0,Y 594.238,Z 668.843,A -85,B 0,C 180,E1 -1259.323,E2 -1259.323} C_VEL
LIN {X 0,Y 594.238,Z 668.863,A -85,B 0,C 180,E1 -1260.678,E2 -1260.678} C_VEL
LIN {X 0,Y 594.229,Z 667.946,A -85,B 0,C 180,E1 -1262.034,E2 -1262.034} C_VEL
LIN {X 0,Y 594.259,Z 666.06,A -85,B 0,C 180,E1 -1263.39,E2 -1263.39} C_VEL
LIN {X 0,Y 594.23,Z 663.175,A -85,B 0,C 180,E1 -1264.749,E2 -1264.749} C_VEL
LIN {X 0,Y 594.255,Z 659.268,A -85,B 0,C 180,E1 -1266.11,E2 -1266.11} C_VEL
LIN {X 0,Y 594.283,Z 654.24,A -85,B 0,C 180,E1 -1267.475,E2 -1267.475} C_VEL
LIN {X 0,Y 594.327,Z 648.079,A -85,B 0,C 180,E1 -1268.843,E2 -1268.843} C_VEL
LIN {X 0,Y 594.359,Z 639.516,A -85,B 0,C 180,E1 -1270.389,E2 -1270.389} C_VEL
LIN {X 0,Y 594.409,Z 629.955,A -85,B 0,C 180,E1 -1271.816,E2 -1271.816} C_VEL
LIN {X 0,Y 594.463,Z 619.322,A -85,B 0,C 180,E1 -1273.155,E2 -1273.155} C_VEL
LIN {X 0,Y 594.537,Z 610.597,A -85,B 0,C 180,E1 -1274.112,E2 -1274.112} C_VEL
LIN {X 0,Y 593.941,Z 606.588,A -85,B 0,C 180,E1 -1274.527,E2 -1274.527} C_VEL
LIN {X 0,Y 588.87,Z 594.851,A -85,B 0,C 180,E1 -1275.737,E2 -1275.737} C_VEL
LIN {X 0,Y 587.909,Z 590.514,A -85,B 0,C 180,E1 -1276.117,E2 -1276.117} C_VEL
LIN {X 0,Y 587.852,Z 588.985,A -85,B 0,C 180,E1 -1276.238,E2 -1276.238} C_VEL
LIN {X 0,Y 588.033,Z 575.229,A -85,B 0,C 180,E1 -1277.238,E2 -1277.238} C_VEL
LIN {X 0,Y 588.187,Z 561.106,A -85,B 0,C 180,E1 -1278.1,E2 -1278.1} C_VEL
LIN {X 0,Y 588.358,Z 545.949,A -85,B 0,C 180,E1 -1278.867,E2 -1278.867} C_VEL
LIN {X 0,Y 588.527,Z 530.755,A -85,B 0,C 180,E1 -1279.489,E2 -1279.489} C_VEL
LIN {X 0,Y 588.676,Z 514.554,A -85,B 0,C 180,E1 -1280.006,E2 -1280.006} C_VEL
LIN {X 0,Y 588.793,Z 497.8,A -85,B 0,C 180,E1 -1280.389,E2 -1280.389} C_VEL
LIN {X 0,Y 588.668,Z 489.551,A -85,B 0,C 180,E1 -1280.528,E2 -1280.528} C_VEL
LIN {X 0,Y 587.355,Z 485.636,A -85,B 0,C 180,E1 -1280.647,E2 -1280.647} C_VEL
LIN {X 0,Y 587.324,Z 485.642,A -85,B 0,C 180,E1 -1283.259,E2 -1283.259} C_VEL
LIN {X 0,Y 587.338,Z 485.636,A -85,B 0,C 180,E1 -1285.517,E2 -1285.517} C_VEL
LIN {X 0,Y 587.343,Z 485.636,A -85,B 0,C 180,E1 -1287.818,E2 -1287.818} C_VEL
LIN {X 0,Y 587.339,Z 485.638,A -85,B 0,C 180,E1 -1290.51,E2 -1290.51} C_VEL
LIN {X 0,Y 587.339,Z 485.638,A -85,B 0,C 180,E1 -1293.397,E2 -1293.397} C_VEL
LIN {X 0,Y 587.351,Z 485.637,A -85,B 0,C 180,E1 -1295.896,E2 -1295.896} C_VEL
LIN {X 0,Y 587.33,Z 485.637,A -85,B 0,C 180,E1 -1298.48,E2 -1298.48} C_VEL
LIN {X 0,Y 587.338,Z 485.636,A -85,B 0,C 180,E1 -1301.157,E2 -1301.157} C_VEL
LIN {X 0,Y 587.317,Z 485.638,A -85,B 0,C 180,E1 -1304.112,E2 -1304.112} C_VEL
LIN {X 0,Y 587.327,Z 485.637,A -85,B 0,C 180,E1 -1306.994,E2 -1306.994} C_VEL
LIN {X 0,Y 587.323,Z 485.637,A -85,B 0,C 180,E1 -1309.746,E2 -1309.746} C_VEL
LIN {X 0,Y 587.349,Z 485.634,A -85,B 0,C 180,E1 -1312.392,E2 -1312.392} C_VEL
LIN {X 0,Y 587.351,Z 485.635,A -85,B 0,C 180,E1 -1315.653,E2 -1315.653} C_VEL
LIN {X 0,Y 587.347,Z 485.635,A -85,B 0,C 180,E1 -1318.231,E2 -1318.231} C_VEL
LIN {X 0,Y 587.352,Z 485.634,A -85,B 0,C 180,E1 -1320.867,E2 -1320.867} C_VEL
LIN {X 0,Y 587.364,Z 485.633,A -85,B 0,C 180,E1 -1323.819,E2 -1323.819} C_VEL
LIN {X 0,Y 587.34,Z 485.722,A -85,B 0,C 180,E1 -1325.993,E2 -1325.993} C_VEL
LIN {X 0,Y 587.337,Z 491.501,A -85,B 0,C 180,E1 -1328.962,E2 -1328.962} C_VEL
LIN {X 0,Y 587.297,Z 496.874,A -85,B 0,C 180,E1 -1331.872,E2 -1331.872} C_VEL
LIN {X 0,Y 587.28,Z 502.288,A -85,B 0,C 180,E1 -1334.735,E2 -1334.735} C_VEL
LIN {X 0,Y 587.253,Z 506.405,A -85,B 0,C 180,E1 -1336.856,E2 -1336.856} C_VEL
LIN {X 0,Y 587.271,Z 511.963,A -85,B 0,C 180,E1 -1339.658,E2 -1339.658} C_VEL
LIN {X 0,Y 587.246,Z 517.603,A -85,B 0,C 180,E1 -1342.435,E2 -1342.435} C_VEL
LIN {X 0,Y 587.219,Z 521.66,A -85,B 0,C 180,E1 -1344.397,E2 -1344.397} C_VEL
LIN {X 0,Y 588.814,Z 527.823,A -85,B 0,C 180,E1 -1344.541,E2 -1344.541} C_VEL
LIN {X 0,Y 588.799,Z 543.714,A -85,B 0,C 180,E1 -1344.82,E2 -1344.82} C_VEL
LIN {X 0,Y 588.619,Z 559.422,A -85,B 0,C 180,E1 -1345.226,E2 -1345.226} C_VEL
LIN {X 0,Y 588.436,Z 576.151,A -85,B 0,C 180,E1 -1345.804,E2 -1345.804} C_VEL
LIN {X 0,Y 588.304,Z 591.559,A -85,B 0,C 180,E1 -1346.489,E2 -1346.489} C_VEL
LIN {X 0,Y 588.126,Z 605.792,A -85,B 0,C 180,E1 -1347.26,E2 -1347.26} C_VEL
LIN {X 0,Y 587.939,Z 619.038,A -85,B 0,C 180,E1 -1348.116,E2 -1348.116} C_VEL
LIN {X 0,Y 587.772,Z 633.606,A -85,B 0,C 180,E1 -1349.229,E2 -1349.229} C_VEL
LIN {X 0,Y 587.623,Z 645.922,A -85,B 0,C 180,E1 -1350.342,E2 -1350.342} C_VEL
LIN {X 0,Y 587.457,Z 657.331,A -85,B 0,C 180,E1 -1351.542,E2 -1351.542} C_VEL
LIN {X 0,Y 587.412,Z 668.406,A -85,B 0,C 180,E1 -1352.914,E2 -1352.914} C_VEL
LIN {X 0,Y 587.301,Z 677.751,A -85,B 0,C 180,E1 -1354.288,E2 -1354.288} C_VEL
LIN {X 0,Y 587.228,Z 684.716,A -85,B 0,C 180,E1 -1355.493,E2 -1355.493} C_VEL
LIN {X 0,Y 587.209,Z 691.5,A -85,B 0,C 180,E1 -1356.873,E2 -1356.873} C_VEL
LIN {X 0,Y 587.187,Z 697.026,A -85,B 0,C 180,E1 -1358.257,E2 -1358.257} C_VEL
LIN {X 0,Y 587.151,Z 701.519,A -85,B 0,C 180,E1 -1359.646,E2 -1359.646} C_VEL
LIN {X 0,Y 587.166,Z 704.875,A -85,B 0,C 180,E1 -1361.04,E2 -1361.04} C_VEL
LIN {X 0,Y 587.154,Z 707.271,A -85,B 0,C 180,E1 -1362.441,E2 -1362.441} C_VEL
LIN {X 0,Y 587.159,Z 708.795,A -85,B 0,C 180,E1 -1364.179,E2 -1364.179} C_VEL
LIN {X 0,Y 587.129,Z 708.772,A -85,B 0,C 180,E1 -1365.98,E2 -1365.98} C_VEL
LIN {X 0,Y 587.128,Z 707.541,A -85,B 0,C 180,E1 -1367.412,E2 -1367.412} C_VEL
LIN {X 0,Y 587.148,Z 705.015,A -85,B 0,C 180,E1 -1368.983,E2 -1368.983} C_VEL
LIN {X 0,Y 587.174,Z 700.896,A -85,B 0,C 180,E1 -1370.653,E2 -1370.653} C_VEL
LIN {X 0,Y 587.175,Z 695.887,A -85,B 0,C 180,E1 -1372.149,E2 -1372.149} C_VEL
LIN {X 0,Y 587.199,Z 689.553,A -85,B 0,C 180,E1 -1373.637,E2 -1373.637} C_VEL
LIN {X 0,Y 587.279,Z 681.698,A -85,B 0,C 180,E1 -1375.139,E2 -1375.139} C_VEL
LIN {X 0,Y 587.333,Z 673.402,A -85,B 0,C 180,E1 -1376.469,E2 -1376.469} C_VEL
LIN {X 0,Y 587.413,Z 663.469,A -85,B 0,C 180,E1 -1377.813,E2 -1377.813} C_VEL
LIN {X 0,Y 587.545,Z 651.689,A -85,B 0,C 180,E1 -1379.167,E2 -1379.167} C_VEL
LIN {X 0,Y 587.703,Z 640.239,A -85,B 0,C 180,E1 -1380.283,E2 -1380.283} C_VEL
LIN {X 0,Y 587.834,Z 627.712,A -85,B 0,C 180,E1 -1381.336,E2 -1381.336} C_VEL
LIN {X 0,Y 588.017,Z 613.691,A -85,B 0,C 180,E1 -1382.34,E2 -1382.34} C_VEL
LIN {X 0,Y 588.227,Z 598.519,A -85,B 0,C 180,E1 -1383.243,E2 -1383.243} C_VEL
LIN {X 0,Y 588.388,Z 583.091,A -85,B 0,C 180,E1 -1383.996,E2 -1383.996} C_VEL
LIN {X 0,Y 588.525,Z 568.167,A -85,B 0,C 180,E1 -1384.582,E2 -1384.582} C_VEL
LIN {X 0,Y 588.711,Z 551.417,A -85,B 0,C 180,E1 -1385.088,E2 -1385.088} C_VEL
LIN {X 0,Y 588.784,Z 535.344,A -85,B 0,C 180,E1 -1385.433,E2 -1385.433} C_VEL
LIN {X 0,Y 588.762,Z 527.589,A -85,B 0,C 180,E1 -1385.554,E2 -1385.554} C_VEL
LIN {X 0,Y 587.232,Z 521.63,A -85,B 0,C 180,E1 -1385.706,E2 -1385.706} C_VEL
LIN {X 0,Y 587.223,Z 515.905,A -85,B 0,C 180,E1 -1388.486,E2 -1388.486} C_VEL
LIN {X 0,Y 587.254,Z 510.502,A -85,B 0,C 180,E1 -1391.162,E2 -1391.162} C_VEL
LIN {X 0,Y 587.265,Z 504.997,A -85,B 0,C 180,E1 -1393.954,E2 -1393.954} C_VEL
LIN {X 0,Y 587.291,Z 499.379,A -85,B 0,C 180,E1 -1396.882,E2 -1396.882} C_VEL
LIN {X 0,Y 587.313,Z 494.056,A -85,B 0,C 180,E1 -1399.745,E2 -1399.745} C_VEL
LIN {X 0,Y 587.331,Z 489.085,A -85,B 0,C 180,E1 -1402.391,E2 -1402.391} C_VEL
LIN {X 0,Y 587.305,Z 485.645,A -85,B 0,C 180,E1 -1404.1,E2 -1404.1} C_VEL
LIN {X 0,Y 587.332,Z 485.641,A -85,B 0,C 180,E1 -1406.603,E2 -1406.603} C_VEL
LIN {X 0,Y 587.343,Z 485.64,A -85,B 0,C 180,E1 -1409.487,E2 -1409.487} C_VEL
LIN {X 0,Y 587.343,Z 485.639,A -85,B 0,C 180,E1 -1412.306,E2 -1412.306} C_VEL
LIN {X 0,Y 587.337,Z 485.637,A -85,B 0,C 180,E1 -1414.483,E2 -1414.483} C_VEL
LIN {X 0,Y 587.362,Z 485.636,A -85,B 0,C 180,E1 -1417.487,E2 -1417.487} C_VEL
LIN {X 0,Y 587.336,Z 485.639,A -85,B 0,C 180,E1 -1420.424,E2 -1420.424} C_VEL
LIN {X 0,Y 587.346,Z 485.636,A -85,B 0,C 180,E1 -1423.311,E2 -1423.311} C_VEL
LIN {X 0,Y 587.354,Z 485.634,A -85,B 0,C 180,E1 -1426.154,E2 -1426.154} C_VEL
LIN {X 0,Y 587.336,Z 485.636,A -85,B 0,C 180,E1 -1428.962,E2 -1428.962} C_VEL
LIN {X 0,Y 587.365,Z 485.632,A -85,B 0,C 180,E1 -1431.744,E2 -1431.744} C_VEL
LIN {X 0,Y 587.361,Z 485.633,A -85,B 0,C 180,E1 -1434.507,E2 -1434.507} C_VEL
LIN {X 0,Y 587.374,Z 485.631,A -85,B 0,C 180,E1 -1437.256,E2 -1437.256} C_VEL
LIN {X 0,Y 587.373,Z 485.632,A -85,B 0,C 180,E1 -1440,E2 -1440} C_VEL
LIN {X 0,Y 587.375,Z 485.631,A -85,B 0,C 180,E1 -1442.743,E2 -1442.743} C_VEL
LIN {X 0,Y 587.351,Z 485.633,A -85,B 0,C 180,E1 -1445.493,E2 -1445.493} C_VEL
LIN {X 0,Y 587.364,Z 485.632,A -85,B 0,C 180,E1 -1448.255,E2 -1448.255} C_VEL
LIN {X 0,Y 587.351,Z 485.635,A -85,B 0,C 180,E1 -1451.141,E2 -1451.141} C_VEL
LIN {X 0,Y 587.354,Z 485.639,A -85,B 0,C 180,E1 -1454.261,E2 -1454.261} C_VEL
LIN {X 0,Y 587.35,Z 485.631,A -85,B 0,C 180,E1 -1457.406,E2 -1457.406} C_VEL
LIN {X 0,Y 587.327,Z 485.637,A -85,B 0,C 180,E1 -1460.305,E2 -1460.305} C_VEL
LIN {X 0,Y 587.358,Z 485.632,A -85,B 0,C 180,E1 -1463.257,E2 -1463.257} C_VEL
LIN {X 0,Y 587.355,Z 485.635,A -85,B 0,C 180,E1 -1466.277,E2 -1466.277} C_VEL
LIN {X 0,Y 587.346,Z 485.639,A -85,B 0,C 180,E1 -1469.135,E2 -1469.135} C_VEL
LIN {X 0,Y 587.349,Z 485.638,A -85,B 0,C 180,E1 -1471.839,E2 -1471.839} C_VEL
LIN {X 0,Y 587.351,Z 485.636,A -85,B 0,C 180,E1 -1474.35,E2 -1474.35} C_VEL
LIN {X 0,Y 587.345,Z 485.635,A -85,B 0,C 180,E1 -1476.747,E2 -1476.747} C_VEL
LIN {X 0,Y 587.342,Z 485.635,A -85,B 0,C 180,E1 -1479.359,E2 -1479.359} C_VEL
LIN {X 0,Y 587.325,Z 485.638,A -85,B 0,C 180,E1 -1482.108,E2 -1482.108} C_VEL
LIN {X 0,Y 587.306,Z 485.641,A -85,B 0,C 180,E1 -1484.912,E2 -1484.912} C_VEL
LIN {X 0,Y 587.344,Z 485.638,A -85,B 0,C 180,E1 -1487.928,E2 -1487.928} C_VEL
LIN {X 0,Y 587.37,Z 485.789,A -85,B 0,C 180,E1 -1489.131,E2 -1489.131} C_VEL
LIN {X 0,Y 588.319,Z 490.301,A -85,B 0,C 180,E1 -1490.325,E2 -1490.325} C_VEL
LIN {X 0,Y 588.224,Z 500.923,A -85,B 0,C 180,E1 -1492.872,E2 -1492.872} C_VEL
LIN {X 0,Y 588.098,Z 512.466,A -85,B 0,C 180,E1 -1495.545,E2 -1495.545} C_VEL
LIN {X 0,Y 587.951,Z 524.612,A -85,B 0,C 180,E1 -1498.269,E2 -1498.269} C_VEL
LIN {X 0,Y 587.833,Z 537.637,A -85,B 0,C 180,E1 -1501.108,E2 -1501.108} C_VEL
LIN {X 0,Y 587.698,Z 550.095,A -85,B 0,C 180,E1 -1503.752,E2 -1503.752} C_VEL
LIN {X 0,Y 587.612,Z 562.754,A -85,B 0,C 180,E1 -1506.381,E2 -1506.381} C_VEL
LIN {X 0,Y 587.525,Z 577.142,A -85,B 0,C 180,E1 -1509.309,E2 -1509.309} C_VEL
LIN {X 0,Y 588.812,Z 582.871,A -85,B 0,C 180,E1 -1509.43,E2 -1509.43} C_VEL
LIN {X 0,Y 588.737,Z 600.112,A -85,B 0,C 180,E1 -1509.701,E2 -1509.701} C_VEL
LIN {X 0,Y 588.642,Z 616.964,A -85,B 0,C 180,E1 -1510.108,E2 -1510.108} C_VEL
LIN {X 0,Y 588.537,Z 632.724,A -85,B 0,C 180,E1 -1510.626,E2 -1510.626} C_VEL
LIN {X 0,Y 588.306,Z 648.063,A -85,B 0,C 180,E1 -1511.274,E2 -1511.274} C_VEL
LIN {X 0,Y 588.148,Z 663.46,A -85,B 0,C 180,E1 -1512.081,E2 -1512.081} C_VEL
LIN {X 0,Y 587.959,Z 677.886,A -85,B 0,C 180,E1 -1512.99,E2 -1512.99} C_VEL
LIN {X 0,Y 587.803,Z 691.864,A -85,B 0,C 180,E1 -1514.039,E2 -1514.039} C_VEL
LIN {X 0,Y 587.671,Z 703.95,A -85,B 0,C 180,E1 -1515.102,E2 -1515.102} C_VEL
LIN {X 0,Y 587.5,Z 715.897,A -85,B 0,C 180,E1 -1516.335,E2 -1516.335} C_VEL
LIN {X 0,Y 587.396,Z 726.06,A -85,B 0,C 180,E1 -1517.564,E2 -1517.564} C_VEL
LIN {X 0,Y 587.334,Z 735.936,A -85,B 0,C 180,E1 -1518.963,E2 -1518.963} C_VEL
LIN {X 0,Y 587.237,Z 744.234,A -85,B 0,C 180,E1 -1520.355,E2 -1520.355} C_VEL
LIN {X 0,Y 587.227,Z 751.108,A -85,B 0,C 180,E1 -1521.744,E2 -1521.744} C_VEL
LIN {X 0,Y 587.203,Z 756.72,A -85,B 0,C 180,E1 -1523.127,E2 -1523.127} C_VEL
LIN {X 0,Y 587.187,Z 761.248,A -85,B 0,C 180,E1 -1524.506,E2 -1524.506} C_VEL
LIN {X 0,Y 587.168,Z 764.635,A -85,B 0,C 180,E1 -1525.882,E2 -1525.882} C_VEL
LIN {X 0,Y 587.12,Z 767.088,A -85,B 0,C 180,E1 -1527.256,E2 -1527.256} C_VEL
LIN {X 0,Y 587.144,Z 768.478,A -85,B 0,C 180,E1 -1528.629,E2 -1528.629} C_VEL
LIN {X 0,Y 587.132,Z 769,A -85,B 0,C 180,E1 -1530.001,E2 -1530.001} C_VEL
LIN {X 0,Y 587.144,Z 768.477,A -85,B 0,C 180,E1 -1531.372,E2 -1531.372} C_VEL
LIN {X 0,Y 587.12,Z 767.085,A -85,B 0,C 180,E1 -1532.745,E2 -1532.745} C_VEL
LIN {X 0,Y 587.168,Z 764.632,A -85,B 0,C 180,E1 -1534.119,E2 -1534.119} C_VEL
LIN {X 0,Y 587.185,Z 760.183,A -85,B 0,C 180,E1 -1535.84,E2 -1535.84} C_VEL
LIN {X 0,Y 587.213,Z 755.466,A -85,B 0,C 180,E1 -1537.22,E2 -1537.22} C_VEL
LIN {X 0,Y 587.245,Z 747.854,A -85,B 0,C 180,E1 -1538.951,E2 -1538.951} C_VEL
LIN {X 0,Y 587.284,Z 739.243,A -85,B 0,C 180,E1 -1540.516,E2 -1540.516} C_VEL
LIN {X 0,Y 587.365,Z 729.965,A -85,B 0,C 180,E1 -1541.912,E2 -1541.912} C_VEL
LIN {X 0,Y 587.45,Z 720.417,A -85,B 0,C 180,E1 -1543.139,E2 -1543.139} C_VEL
LIN {X 0,Y 587.563,Z 709.628,A -85,B 0,C 180,E1 -1544.336,E2 -1544.336} C_VEL
LIN {X 0,Y 587.74,Z 697.136,A -85,B 0,C 180,E1 -1545.519,E2 -1545.519} C_VEL
LIN {X 0,Y 587.91,Z 682.702,A -85,B 0,C 180,E1 -1546.673,E2 -1546.673} C_VEL
LIN {X 0,Y 588.089,Z 668.006,A -85,B 0,C 180,E1 -1547.653,E2 -1547.653} C_VEL
LIN {X 0,Y 588.252,Z 653.505,A -85,B 0,C 180,E1 -1548.458,E2 -1548.458} C_VEL
LIN {X 0,Y 588.468,Z 637.509,A -85,B 0,C 180,E1 -1549.184,E2 -1549.184} C_VEL
LIN {X 0,Y 588.617,Z 621.465,A -85,B 0,C 180,E1 -1549.758,E2 -1549.758} C_VEL
LIN {X 0,Y 588.755,Z 604.594,A -85,B 0,C 180,E1 -1550.208,E2 -1550.208} C_VEL
LIN {X 0,Y 588.819,Z 587.88,A -85,B 0,C 180,E1 -1550.503,E2 -1550.503} C_VEL
LIN {X 0,Y 588.577,Z 581.409,A -85,B 0,C 180,E1 -1550.597,E2 -1550.597} C_VEL
LIN {X 0,Y 587.511,Z 577.049,A -85,B 0,C 180,E1 -1550.71,E2 -1550.71} C_VEL
LIN {X 0,Y 587.614,Z 562.746,A -85,B 0,C 180,E1 -1553.62,E2 -1553.62} C_VEL
LIN {X 0,Y 587.746,Z 548.216,A -85,B 0,C 180,E1 -1556.642,E2 -1556.642} C_VEL
LIN {X 0,Y 587.847,Z 535.502,A -85,B 0,C 180,E1 -1559.353,E2 -1559.353} C_VEL
LIN {X 0,Y 587.974,Z 522.558,A -85,B 0,C 180,E1 -1562.186,E2 -1562.186} C_VEL
LIN {X 0,Y 588.1,Z 511.49,A -85,B 0,C 180,E1 -1564.678,E2 -1564.678} C_VEL
LIN {X 0,Y 588.268,Z 499.177,A -85,B 0,C 180,E1 -1567.539,E2 -1567.539} C_VEL
LIN {X 0,Y 588.316,Z 490.296,A -85,B 0,C 180,E1 -1569.677,E2 -1569.677} C_VEL
LIN {X 0,Y 587.353,Z 485.639,A -85,B 0,C 180,E1 -1570.929,E2 -1570.929} C_VEL
LIN {X 0,Y 587.336,Z 485.633,A -85,B 0,C 180,E1 -1573.95,E2 -1573.95} C_VEL
LIN {X 0,Y 587.326,Z 485.641,A -85,B 0,C 180,E1 -1576.881,E2 -1576.881} C_VEL
LIN {X 0,Y 587.319,Z 485.634,A -85,B 0,C 180,E1 -1579.746,E2 -1579.746} C_VEL
LIN {X 0,Y 587.344,Z 485.639,A -85,B 0,C 180,E1 -1582.393,E2 -1582.393} C_VEL
LIN {X 0,Y 587.337,Z 485.634,A -85,B 0,C 180,E1 -1584.945,E2 -1584.945} C_VEL
LIN {X 0,Y 587.338,Z 485.632,A -85,B 0,C 180,E1 -1587.421,E2 -1587.421} C_VEL
LIN {X 0,Y 587.335,Z 485.636,A -85,B 0,C 180,E1 -1589.83,E2 -1589.83} C_VEL
LIN {X 0,Y 587.353,Z 485.636,A -85,B 0,C 180,E1 -1592.307,E2 -1592.307} C_VEL
LIN {X 0,Y 587.337,Z 485.635,A -85,B 0,C 180,E1 -1594.484,E2 -1594.484} C_VEL
LIN {X 0,Y 587.319,Z 485.635,A -85,B 0,C 180,E1 -1597.132,E2 -1597.132} C_VEL
LIN {X 0,Y 587.355,Z 485.635,A -85,B 0,C 180,E1 -1599.456,E2 -1599.456} C_VEL
LIN {X 0,Y 588.805,Z 489.836,A -85,B 0,C 180,E1 -1599.571,E2 -1599.571} C_VEL
LIN {X 0,Y 588.707,Z 506.597,A -85,B 0,C 180,E1 -1599.882,E2 -1599.882} C_VEL
LIN {X 0,Y 588.615,Z 523.012,A -85,B 0,C 180,E1 -1600.333,E2 -1600.333} C_VEL
LIN {X 0,Y 588.437,Z 539.473,A -85,B 0,C 180,E1 -1600.939,E2 -1600.939} C_VEL
LIN {X 0,Y 588.241,Z 554.418,A -85,B 0,C 180,E1 -1601.633,E2 -1601.633} C_VEL
LIN {X 0,Y 588.126,Z 568.735,A -85,B 0,C 180,E1 -1602.439,E2 -1602.439} C_VEL
LIN {X 0,Y 587.909,Z 583.299,A -85,B 0,C 180,E1 -1603.417,E2 -1603.417} C_VEL
LIN {X 0,Y 587.734,Z 596.616,A -85,B 0,C 180,E1 -1604.481,E2 -1604.481} C_VEL
LIN {X 0,Y 587.566,Z 609.18,A -85,B 0,C 180,E1 -1605.664,E2 -1605.664} C_VEL
LIN {X 0,Y 587.45,Z 620.056,A -85,B 0,C 180,E1 -1606.862,E2 -1606.862} C_VEL
LIN {X 0,Y 587.359,Z 630.899,A -85,B 0,C 180,E1 -1608.264,E2 -1608.264} C_VEL
LIN {X 0,Y 587.299,Z 640.008,A -85,B 0,C 180,E1 -1609.66,E2 -1609.66} C_VEL
LIN {X 0,Y 587.248,Z 647.627,A -85,B 0,C 180,E1 -1611.05,E2 -1611.05} C_VEL
LIN {X 0,Y 587.202,Z 653.869,A -85,B 0,C 180,E1 -1612.435,E2 -1612.435} C_VEL
LIN {X 0,Y 587.16,Z 658.993,A -85,B 0,C 180,E1 -1613.816,E2 -1613.816} C_VEL
LIN {X 0,Y 587.133,Z 662.948,A -85,B 0,C 180,E1 -1615.194,E2 -1615.194} C_VEL
LIN {X 0,Y 587.176,Z 665.916,A -85,B 0,C 180,E1 -1616.569,E2 -1616.569} C_VEL
LIN {X 0,Y 587.129,Z 667.846,A -85,B 0,C 180,E1 -1617.942,E2 -1617.942} C_VEL
LIN {X 0,Y 587.139,Z 668.844,A -85,B 0,C 180,E1 -1619.314,E2 -1619.314} C_VEL
LIN {X 0,Y 587.138,Z 668.865,A -85,B 0,C 180,E1 -1620.686,E2 -1620.686} C_VEL
LIN {X 0,Y 587.128,Z 667.948,A -85,B 0,C 180,E1 -1622.058,E2 -1622.058} C_VEL
LIN {X 0,Y 587.181,Z 666.062,A -85,B 0,C 180,E1 -1623.431,E2 -1623.431} C_VEL
LIN {X 0,Y 587.132,Z 663.175,A -85,B 0,C 180,E1 -1624.807,E2 -1624.807} C_VEL
LIN {X 0,Y 587.164,Z 659.269,A -85,B 0,C 180,E1 -1626.184,E2 -1626.184} C_VEL
LIN {X 0,Y 587.203,Z 654.24,A -85,B 0,C 180,E1 -1627.566,E2 -1627.566} C_VEL
LIN {X 0,Y 587.251,Z 648.077,A -85,B 0,C 180,E1 -1628.951,E2 -1628.951} C_VEL
LIN {X 0,Y 587.284,Z 639.516,A -85,B 0,C 180,E1 -1630.516,E2 -1630.516} C_VEL
LIN {X 0,Y 587.366,Z 630.291,A -85,B 0,C 180,E1 -1631.912,E2 -1631.912} C_VEL
LIN {X 0,Y 587.456,Z 619.32,A -85,B 0,C 180,E1 -1633.315,E2 -1633.315} C_VEL
LIN {X 0,Y 587.592,Z 607.968,A -85,B 0,C 180,E1 -1634.547,E2 -1634.547} C_VEL
LIN {X 0,Y 587.742,Z 595.57,A -85,B 0,C 180,E1 -1635.697,E2 -1635.697} C_VEL
LIN {X 0,Y 587.852,Z 588.985,A -85,B 0,C 180,E1 -1636.238,E2 -1636.238} C_VEL
LIN {X 0,Y 587.277,Z 584.493,A -85,B 0,C 180,E1 -1636.602,E2 -1636.602} C_VEL
LIN {X 0,Y 581.919,Z 569.689,A -85,B 0,C 180,E1 -1637.79,E2 -1637.79} C_VEL
LIN {X 0,Y 581.323,Z 564.775,A -85,B 0,C 180,E1 -1638.107,E2 -1638.107} C_VEL
LIN {X 0,Y 581.512,Z 550.872,A -85,B 0,C 180,E1 -1638.863,E2 -1638.863} C_VEL
LIN {X 0,Y 581.775,Z 534.939,A -85,B 0,C 180,E1 -1639.565,E2 -1639.565} C_VEL
LIN {X 0,Y 581.954,Z 519.143,A -85,B 0,C 180,E1 -1640.109,E2 -1640.109} C_VEL
LIN {X 0,Y 582.105,Z 503.517,A -85,B 0,C 180,E1 -1640.516,E2 -1640.516} C_VEL
LIN {X 0,Y 581.993,Z 491.166,A -85,B 0,C 180,E1 -1640.749,E2 -1640.749} C_VEL
LIN {X 0,Y 580.306,Z 486.513,A -85,B 0,C 180,E1 -1640.892,E2 -1640.892} C_VEL
LIN {X 0,Y 580.281,Z 486.516,A -85,B 0,C 180,E1 -1643.558,E2 -1643.558} C_VEL
LIN {X 0,Y 580.297,Z 486.516,A -85,B 0,C 180,E1 -1645.849,E2 -1645.849} C_VEL
LIN {X 0,Y 580.3,Z 486.512,A -85,B 0,C 180,E1 -1648.186,E2 -1648.186} C_VEL
LIN {X 0,Y 580.287,Z 486.515,A -85,B 0,C 180,E1 -1650.695,E2 -1650.695} C_VEL
LIN {X 0,Y 580.308,Z 486.515,A -85,B 0,C 180,E1 -1653.317,E2 -1653.317} C_VEL
LIN {X 0,Y 580.317,Z 486.512,A -85,B 0,C 180,E1 -1655.766,E2 -1655.766} C_VEL
LIN {X 0,Y 580.29,Z 486.513,A -85,B 0,C 180,E1 -1658.147,E2 -1658.147} C_VEL
LIN {X 0,Y 580.302,Z 486.512,A -85,B 0,C 180,E1 -1660.844,E2 -1660.844} C_VEL
LIN {X 0,Y 580.278,Z 486.516,A -85,B 0,C 180,E1 -1663.658,E2 -1663.658} C_VEL
LIN {X 0,Y 580.291,Z 486.513,A -85,B 0,C 180,E1 -1666.608,E2 -1666.608} C_VEL
LIN {X 0,Y 580.305,Z 486.514,A -85,B 0,C 180,E1 -1669.157,E2 -1669.157} C_VEL
LIN {X 0,Y 580.294,Z 486.516,A -85,B 0,C 180,E1 -1671.927,E2 -1671.927} C_VEL
LIN {X 0,Y 580.256,Z 486.521,A -85,B 0,C 180,E1 -1674.453,E2 -1674.453} C_VEL
LIN {X 0,Y 580.296,Z 486.514,A -85,B 0,C 180,E1 -1676.975,E2 -1676.975} C_VEL
LIN {X 0,Y 580.302,Z 486.513,A -85,B 0,C 180,E1 -1679.425,E2 -1679.425} C_VEL
LIN {X 0,Y 580.303,Z 486.513,A -85,B 0,C 180,E1 -1682.141,E2 -1682.141} C_VEL
LIN {X 0,Y 580.328,Z 486.51,A -85,B 0,C 180,E1 -1685.269,E2 -1685.269} C_VEL
LIN {X 0,Y 580.292,Z 486.7,A -85,B 0,C 180,E1 -1686.063,E2 -1686.063} C_VEL
LIN {X 0,Y 580.287,Z 492.098,A -85,B 0,C 180,E1 -1688.839,E2 -1688.839} C_VEL
LIN {X 0,Y 580.246,Z 497.292,A -85,B 0,C 180,E1 -1691.644,E2 -1691.644} C_VEL
LIN {X 0,Y 580.226,Z 502.7,A -85,B 0,C 180,E1 -1694.545,E2 -1694.545} C_VEL
LIN {X 0,Y 580.198,Z 506.813,A -85,B 0,C 180,E1 -1696.694,E2 -1696.694} C_VEL
LIN {X 0,Y 580.196,Z 512.368,A -85,B 0,C 180,E1 -1699.531,E2 -1699.531} C_VEL
LIN {X 0,Y 580.171,Z 518.005,A -85,B 0,C 180,E1 -1702.342,E2 -1702.342} C_VEL
LIN {X 0,Y 580.163,Z 521.657,A -85,B 0,C 180,E1 -1704.133,E2 -1704.133} C_VEL
LIN {X 0,Y 582.147,Z 529.834,A -85,B 0,C 180,E1 -1704.327,E2 -1704.327} C_VEL
LIN {X 0,Y 582.076,Z 545.071,A -85,B 0,C 180,E1 -1704.608,E2 -1704.608} C_VEL
LIN {X 0,Y 581.921,Z 560.432,A -85,B 0,C 180,E1 -1705.019,E2 -1705.019} C_VEL
LIN {X 0,Y 581.719,Z 576.379,A -85,B 0,C 180,E1 -1705.582,E2 -1705.582} C_VEL
LIN {X 0,Y 581.511,Z 591.752,A -85,B 0,C 180,E1 -1706.275,E2 -1706.275} C_VEL
LIN {X 0,Y 581.297,Z 605.953,A -85,B 0,C 180,E1 -1707.054,E2 -1707.054} C_VEL
LIN {X 0,Y 581.084,Z 619.182,A -85,B 0,C 180,E1 -1707.92,E2 -1707.92} C_VEL
LIN {X 0,Y 580.861,Z 633.737,A -85,B 0,C 180,E1 -1709.046,E2 -1709.046} C_VEL
LIN {X 0,Y 580.649,Z 646.033,A -85,B 0,C 180,E1 -1710.173,E2 -1710.173} C_VEL
LIN {X 0,Y 580.486,Z 657.414,A -85,B 0,C 180,E1 -1711.387,E2 -1711.387} C_VEL
LIN {X 0,Y 580.382,Z 668.485,A -85,B 0,C 180,E1 -1712.776,E2 -1712.776} C_VEL
LIN {X 0,Y 580.247,Z 677.822,A -85,B 0,C 180,E1 -1714.167,E2 -1714.167} C_VEL
LIN {X 0,Y 580.154,Z 685.669,A -85,B 0,C 180,E1 -1715.561,E2 -1715.561} C_VEL
LIN {X 0,Y 580.14,Z 692.297,A -85,B 0,C 180,E1 -1716.957,E2 -1716.957} C_VEL
LIN {X 0,Y 580.109,Z 697.68,A -85,B 0,C 180,E1 -1718.358,E2 -1718.358} C_VEL
LIN {X 0,Y 580.057,Z 702.01,A -85,B 0,C 180,E1 -1719.765,E2 -1719.765} C_VEL
LIN {X 0,Y 580.075,Z 705.26,A -85,B 0,C 180,E1 -1721.177,E2 -1721.177} C_VEL
LIN {X 0,Y 580.044,Z 707.483,A -85,B 0,C 180,E1 -1722.596,E2 -1722.596} C_VEL
LIN {X 0,Y 580.048,Z 708.811,A -85,B 0,C 180,E1 -1724.233,E2 -1724.233} C_VEL
LIN {X 0,Y 580.012,Z 708.913,A -85,B 0,C 180,E1 -1725.46,E2 -1725.46} C_VEL
LIN {X 0,Y 580.038,Z 708.122,A -85,B 0,C 180,E1 -1726.905,E2 -1726.905} C_VEL
LIN {X 0,Y 580.033,Z 706.223,A -85,B 0,C 180,E1 -1728.362,E2 -1728.362} C_VEL
LIN {X 0,Y 580.056,Z 703.271,A -85,B 0,C 180,E1 -1729.83,E2 -1729.83} C_VEL
LIN {X 0,Y 580.082,Z 699.103,A -85,B 0,C 180,E1 -1731.312,E2 -1731.312} C_VEL
LIN {X 0,Y 580.115,Z 692.99,A -85,B 0,C 180,E1 -1732.966,E2 -1732.966} C_VEL
LIN {X 0,Y 580.177,Z 685.744,A -85,B 0,C 180,E1 -1734.515,E2 -1734.515} C_VEL
LIN {X 0,Y 580.256,Z 678.28,A -85,B 0,C 180,E1 -1735.85,E2 -1735.85} C_VEL
LIN {X 0,Y 580.365,Z 667.867,A -85,B 0,C 180,E1 -1737.397,E2 -1737.397} C_VEL
LIN {X 0,Y 580.51,Z 656.871,A -85,B 0,C 180,E1 -1738.765,E2 -1738.765} C_VEL
LIN {X 0,Y 580.664,Z 645.705,A -85,B 0,C 180,E1 -1739.95,E2 -1739.95} C_VEL
LIN {X 0,Y 580.861,Z 634.018,A -85,B 0,C 180,E1 -1741.02,E2 -1741.02} C_VEL
LIN {X 0,Y 581.073,Z 619.454,A -85,B 0,C 180,E1 -1742.151,E2 -1742.151} C_VEL
LIN {X 0,Y 581.296,Z 605.945,A -85,B 0,C 180,E1 -1743.037,E2 -1743.037} C_VEL
LIN {X 0,Y 581.538,Z 590.559,A -85,B 0,C 180,E1 -1743.877,E2 -1743.877} C_VEL
LIN {X 0,Y 581.744,Z 574.212,A -85,B 0,C 180,E1 -1744.596,E2 -1744.596} C_VEL
LIN {X 0,Y 581.915,Z 558.444,A -85,B 0,C 180,E1 -1745.131,E2 -1745.131} C_VEL
LIN {X 0,Y 582.11,Z 542.067,A -85,B 0,C 180,E1 -1745.547,E2 -1745.547} C_VEL
LIN {X 0,Y 582.007,Z 528.462,A -85,B 0,C 180,E1 -1745.79,E2 -1745.79} C_VEL
LIN {X 0,Y 580.121,Z 521.629,A -85,B 0,C 180,E1 -1745.972,E2 -1745.972} C_VEL
LIN {X 0,Y 580.16,Z 515.395,A -85,B 0,C 180,E1 -1749.043,E2 -1749.043} C_VEL
LIN {X 0,Y 580.193,Z 509.971,A -85,B 0,C 180,E1 -1751.775,E2 -1751.775} C_VEL
LIN {X 0,Y 580.203,Z 504.442,A -85,B 0,C 180,E1 -1754.63,E2 -1754.63} C_VEL
LIN {X 0,Y 580.233,Z 499.429,A -85,B 0,C 180,E1 -1757.289,E2 -1757.289} C_VEL
LIN {X 0,Y 580.263,Z 494.298,A -85,B 0,C 180,E1 -1760.064,E2 -1760.064} C_VEL
LIN {X 0,Y 580.277,Z 489.276,A -85,B 0,C 180,E1 -1762.73,E2 -1762.73} C_VEL
LIN {X 0,Y 580.271,Z 486.521,A -85,B 0,C 180,E1 -1764.12,E2 -1764.12} C_VEL
LIN {X 0,Y 580.3,Z 486.518,A -85,B 0,C 180,E1 -1766.682,E2 -1766.682} C_VEL
LIN {X 0,Y 580.302,Z 486.517,A -85,B 0,C 180,E1 -1769.425,E2 -1769.425} C_VEL
LIN {X 0,Y 580.312,Z 486.516,A -85,B 0,C 180,E1 -1772.136,E2 -1772.136} C_VEL
LIN {X 0,Y 580.303,Z 486.517,A -85,B 0,C 180,E1 -1774.92,E2 -1774.92} C_VEL
LIN {X 0,Y 580.321,Z 486.511,A -85,B 0,C 180,E1 -1777.198,E2 -1777.198} C_VEL
LIN {X 0,Y 580.298,Z 486.516,A -85,B 0,C 180,E1 -1780.177,E2 -1780.177} C_VEL
LIN {X 0,Y 580.32,Z 486.513,A -85,B 0,C 180,E1 -1783.103,E2 -1783.103} C_VEL
LIN {X 0,Y 580.318,Z 486.512,A -85,B 0,C 180,E1 -1785.983,E2 -1785.983} C_VEL
LIN {X 0,Y 580.321,Z 486.51,A -85,B 0,C 180,E1 -1788.827,E2 -1788.827} C_VEL
LIN {X 0,Y 580.329,Z 486.509,A -85,B 0,C 180,E1 -1791.644,E2 -1791.644} C_VEL
LIN {X 0,Y 580.328,Z 486.509,A -85,B 0,C 180,E1 -1794.44,E2 -1794.44} C_VEL
LIN {X 0,Y 580.34,Z 486.508,A -85,B 0,C 180,E1 -1797.223,E2 -1797.223} C_VEL
LIN {X 0,Y 580.342,Z 486.507,A -85,B 0,C 180,E1 -1800,E2 -1800} C_VEL
LIN {X 0,Y 580.34,Z 486.507,A -85,B 0,C 180,E1 -1802.776,E2 -1802.776} C_VEL
LIN {X 0,Y 580.317,Z 486.509,A -85,B 0,C 180,E1 -1805.56,E2 -1805.56} C_VEL
LIN {X 0,Y 580.327,Z 486.509,A -85,B 0,C 180,E1 -1808.356,E2 -1808.356} C_VEL
LIN {X 0,Y 580.322,Z 486.511,A -85,B 0,C 180,E1 -1811.208,E2 -1811.208} C_VEL
LIN {X 0,Y 580.316,Z 486.512,A -85,B 0,C 180,E1 -1814.017,E2 -1814.017} C_VEL
LIN {X 0,Y 580.303,Z 486.513,A -85,B 0,C 180,E1 -1816.915,E2 -1816.915} C_VEL
LIN {X 0,Y 580.299,Z 486.516,A -85,B 0,C 180,E1 -1819.822,E2 -1819.822} C_VEL
LIN {X 0,Y 580.319,Z 486.51,A -85,B 0,C 180,E1 -1822.801,E2 -1822.801} C_VEL
LIN {X 0,Y 580.302,Z 486.511,A -85,B 0,C 180,E1 -1825.08,E2 -1825.08} C_VEL
LIN {X 0,Y 580.31,Z 486.516,A -85,B 0,C 180,E1 -1827.864,E2 -1827.864} C_VEL
LIN {X 0,Y 580.289,Z 486.517,A -85,B 0,C 180,E1 -1830.698,E2 -1830.698} C_VEL
LIN {X 0,Y 580.297,Z 486.517,A -85,B 0,C 180,E1 -1833.318,E2 -1833.318} C_VEL
LIN {X 0,Y 580.32,Z 486.512,A -85,B 0,C 180,E1 -1835.769,E2 -1835.769} C_VEL
LIN {X 0,Y 580.28,Z 486.515,A -85,B 0,C 180,E1 -1838.147,E2 -1838.147} C_VEL
LIN {X 0,Y 580.313,Z 486.511,A -85,B 0,C 180,E1 -1840.842,E2 -1840.842} C_VEL
LIN {X 0,Y 580.279,Z 486.516,A -85,B 0,C 180,E1 -1843.658,E2 -1843.658} C_VEL
LIN {X 0,Y 580.284,Z 486.518,A -85,B 0,C 180,E1 -1846.608,E2 -1846.608} C_VEL
LIN {X 0,Y 580.33,Z 486.565,A -85,B 0,C 180,E1 -1848.725,E2 -1848.725} C_VEL
LIN {X 0,Y 581.466,Z 491.919,A -85,B 0,C 180,E1 -1850.165,E2 -1850.165} C_VEL
LIN {X 0,Y 581.454,Z 501.001,A -85,B 0,C 180,E1 -1852.384,E2 -1852.384} C_VEL
LIN {X 0,Y 581.264,Z 513.714,A -85,B 0,C 180,E1 -1855.372,E2 -1855.372} C_VEL
LIN {X 0,Y 581.058,Z 526.428,A -85,B 0,C 180,E1 -1858.256,E2 -1858.256} C_VEL
LIN {X 0,Y 580.925,Z 538.04,A -85,B 0,C 180,E1 -1860.819,E2 -1860.819} C_VEL
LIN {X 0,Y 580.768,Z 550.831,A -85,B 0,C 180,E1 -1863.571,E2 -1863.571} C_VEL
LIN {X 0,Y 580.648,Z 564.57,A -85,B 0,C 180,E1 -1866.459,E2 -1866.459} C_VEL
LIN {X 0,Y 580.508,Z 577.117,A -85,B 0,C 180,E1 -1869.042,E2 -1869.042} C_VEL
LIN {X 0,Y 582.17,Z 584.259,A -85,B 0,C 180,E1 -1869.203,E2 -1869.203} C_VEL
LIN {X 0,Y 582.076,Z 601.316,A -85,B 0,C 180,E1 -1869.483,E2 -1869.483} C_VEL
LIN {X 0,Y 581.953,Z 618.482,A -85,B 0,C 180,E1 -1869.915,E2 -1869.915} C_VEL
LIN {X 0,Y 581.747,Z 634.697,A -85,B 0,C 180,E1 -1870.471,E2 -1870.471} C_VEL
LIN {X 0,Y 581.521,Z 650.013,A -85,B 0,C 180,E1 -1871.139,E2 -1871.139} C_VEL
LIN {X 0,Y 581.335,Z 665.028,A -85,B 0,C 180,E1 -1871.954,E2 -1871.954} C_VEL
LIN {X 0,Y 581.091,Z 678.63,A -85,B 0,C 180,E1 -1872.835,E2 -1872.835} C_VEL
LIN {X 0,Y 580.878,Z 692.925,A -85,B 0,C 180,E1 -1873.934,E2 -1873.934} C_VEL
LIN {X 0,Y 580.692,Z 705.739,A -85,B 0,C 180,E1 -1875.098,E2 -1875.098} C_VEL
LIN {X 0,Y 580.508,Z 717.451,A -85,B 0,C 180,E1 -1876.346,E2 -1876.346} C_VEL
LIN {X 0,Y 580.347,Z 728.737,A -85,B 0,C 180,E1 -1877.766,E2 -1877.766} C_VEL
LIN {X 0,Y 580.239,Z 738.178,A -85,B 0,C 180,E1 -1879.18,E2 -1879.18} C_VEL
LIN {X 0,Y 580.16,Z 746.052,A -85,B 0,C 180,E1 -1880.589,E2 -1880.589} C_VEL
LIN {X 0,Y 580.141,Z 752.628,A -85,B 0,C 180,E1 -1881.993,E2 -1881.993} C_VEL
LIN {X 0,Y 580.125,Z 758.027,A -85,B 0,C 180,E1 -1883.411,E2 -1883.411} C_VEL
LIN {X 0,Y 580.111,Z 761.248,A -85,B 0,C 180,E1 -1884.439,E2 -1884.439} C_VEL
LIN {X 0,Y 580.086,Z 764.636,A -85,B 0,C 180,E1 -1885.832,E2 -1885.832} C_VEL
LIN {X 0,Y 580.031,Z 767.088,A -85,B 0,C 180,E1 -1887.223,E2 -1887.223} C_VEL
LIN {X 0,Y 580.044,Z 768.478,A -85,B 0,C 180,E1 -1888.612,E2 -1888.612} C_VEL
LIN {X 0,Y 580.033,Z 769,A -85,B 0,C 180,E1 -1890.001,E2 -1890.001} C_VEL
LIN {X 0,Y 580.044,Z 768.477,A -85,B 0,C 180,E1 -1891.389,E2 -1891.389} C_VEL
LIN {X 0,Y 580.031,Z 767.086,A -85,B 0,C 180,E1 -1892.779,E2 -1892.779} C_VEL
LIN {X 0,Y 580.086,Z 764.632,A -85,B 0,C 180,E1 -1894.169,E2 -1894.169} C_VEL
LIN {X 0,Y 580.096,Z 760.184,A -85,B 0,C 180,E1 -1895.911,E2 -1895.911} C_VEL
LIN {X 0,Y 580.123,Z 755.466,A -85,B 0,C 180,E1 -1897.309,E2 -1897.309} C_VEL
LIN {X 0,Y 580.179,Z 747.854,A -85,B 0,C 180,E1 -1899.061,E2 -1899.061} C_VEL
LIN {X 0,Y 580.209,Z 739.244,A -85,B 0,C 180,E1 -1900.645,E2 -1900.645} C_VEL
LIN {X 0,Y 580.335,Z 729.965,A -85,B 0,C 180,E1 -1902.059,E2 -1902.059} C_VEL
LIN {X 0,Y 580.441,Z 720.418,A -85,B 0,C 180,E1 -1903.301,E2 -1903.301} C_VEL
LIN {X 0,Y 580.624,Z 708.925,A -85,B 0,C 180,E1 -1904.582,E2 -1904.582} C_VEL
LIN {X 0,Y 580.814,Z 697.136,A -85,B 0,C 180,E1 -1905.709,E2 -1905.709} C_VEL
LIN {X 0,Y 581.012,Z 683.876,A -85,B 0,C 180,E1 -1906.786,E2 -1906.786} C_VEL
LIN {X 0,Y 581.247,Z 669.424,A -85,B 0,C 180,E1 -1907.777,E2 -1907.777} C_VEL
LIN {X 0,Y 581.437,Z 655.254,A -85,B 0,C 180,E1 -1908.591,E2 -1908.591} C_VEL
LIN {X 0,Y 581.677,Z 640.137,A -85,B 0,C 180,E1 -1909.309,E2 -1909.309} C_VEL
LIN {X 0,Y 581.908,Z 624.331,A -85,B 0,C 180,E1 -1909.904,E2 -1909.904} C_VEL
LIN {X 0,Y 582.04,Z 608.328,A -85,B 0,C 180,E1 -1910.36,E2 -1910.36} C_VEL
LIN {X 0,Y 582.141,Z 593.083,A -85,B 0,C 180,E1 -1910.669,E2 -1910.669} C_VEL
LIN {X 0,Y 582.022,Z 583.022,A -85,B 0,C 180,E1 -1910.819,E2 -1910.819} C_VEL
LIN {X 0,Y 580.51,Z 577.112,A -85,B 0,C 180,E1 -1910.959,E2 -1910.959} C_VEL
LIN {X 0,Y 580.651,Z 564.562,A -85,B 0,C 180,E1 -1913.542,E2 -1913.542} C_VEL
LIN {X 0,Y 580.806,Z 550.032,A -85,B 0,C 180,E1 -1916.598,E2 -1916.598} C_VEL
LIN {X 0,Y 580.942,Z 536.932,A -85,B 0,C 180,E1 -1919.422,E2 -1919.422} C_VEL
LIN {X 0,Y 581.097,Z 524.584,A -85,B 0,C 180,E1 -1922.156,E2 -1922.156} C_VEL
LIN {X 0,Y 581.273,Z 513.411,A -85,B 0,C 180,E1 -1924.698,E2 -1924.698} C_VEL
LIN {X 0,Y 581.458,Z 500.993,A -85,B 0,C 180,E1 -1927.618,E2 -1927.618} C_VEL
LIN {X 0,Y 581.468,Z 491.911,A -85,B 0,C 180,E1 -1929.836,E2 -1929.836} C_VEL
LIN {X 0,Y 580.287,Z 486.516,A -85,B 0,C 180,E1 -1931.332,E2 -1931.332} C_VEL
LIN {X 0,Y 580.29,Z 486.511,A -85,B 0,C 180,E1 -1933.657,E2 -1933.657} C_VEL
LIN {X 0,Y 580.286,Z 486.518,A -85,B 0,C 180,E1 -1936.609,E2 -1936.609} C_VEL
LIN {X 0,Y 580.301,Z 486.511,A -85,B 0,C 180,E1 -1939.157,E2 -1939.157} C_VEL
LIN {X 0,Y 580.29,Z 486.512,A -85,B 0,C 180,E1 -1941.927,E2 -1941.927} C_VEL
LIN {X 0,Y 580.3,Z 486.517,A -85,B 0,C 180,E1 -1944.456,E2 -1944.456} C_VEL
LIN {X 0,Y 580.292,Z 486.511,A -85,B 0,C 180,E1 -1946.976,E2 -1946.976} C_VEL
LIN {X 0,Y 580.296,Z 486.509,A -85,B 0,C 180,E1 -1949.425,E2 -1949.425} C_VEL
LIN {X 0,Y 580.321,Z 486.514,A -85,B 0,C 180,E1 -1952.137,E2 -1952.137} C_VEL
LIN {X 0,Y 580.323,Z 486.507,A -85,B 0,C 180,E1 -1955.27,E2 -1955.27} C_VEL
LIN {X 0,Y 580.276,Z 486.52,A -85,B 0,C 180,E1 -1957.948,E2 -1957.948} C_VEL
LIN {X 0,Y 580.315,Z 486.51,A -85,B 0,C 180,E1 -1959.202,E2 -1959.202} C_VEL
LIN {X 0,Y 582.127,Z 491.441,A -85,B 0,C 180,E1 -1959.349,E2 -1959.349} C_VEL
LIN {X 0,Y 582.034,Z 508.457,A -85,B 0,C 180,E1 -1959.687,E2 -1959.687} C_VEL
LIN {X 0,Y 581.881,Z 524.398,A -85,B 0,C 180,E1 -1960.142,E2 -1960.142} C_VEL
LIN {X 0,Y 581.682,Z 540.914,A -85,B 0,C 180,E1 -1960.768,E2 -1960.768} C_VEL
LIN {X 0,Y 581.434,Z 556.183,A -85,B 0,C 180,E1 -1961.501,E2 -1961.501} C_VEL
LIN {X 0,Y 581.23,Z 571.568,A -85,B 0,C 180,E1 -1962.405,E2 -1962.405} C_VEL
LIN {X 0,Y 581.019,Z 585.655,A -85,B 0,C 180,E1 -1963.396,E2 -1963.396} C_VEL
LIN {X 0,Y 580.79,Z 597.648,A -85,B 0,C 180,E1 -1964.381,E2 -1964.381} C_VEL
LIN {X 0,Y 580.582,Z 609.903,A -85,B 0,C 180,E1 -1965.56,E2 -1965.56} C_VEL
LIN {X 0,Y 580.445,Z 621.554,A -85,B 0,C 180,E1 -1966.878,E2 -1966.878} C_VEL
LIN {X 0,Y 580.308,Z 632.146,A -85,B 0,C 180,E1 -1968.296,E2 -1968.296} C_VEL
LIN {X 0,Y 580.24,Z 641.026,A -85,B 0,C 180,E1 -1969.709,E2 -1969.709} C_VEL
LIN {X 0,Y 580.167,Z 649.29,A -85,B 0,C 180,E1 -1971.291,E2 -1971.291} C_VEL
LIN {X 0,Y 580.124,Z 655.295,A -85,B 0,C 180,E1 -1972.692,E2 -1972.692} C_VEL
LIN {X 0,Y 580.114,Z 661.118,A -85,B 0,C 180,E1 -1974.439,E2 -1974.439} C_VEL
LIN {X 0,Y 580.085,Z 664.544,A -85,B 0,C 180,E1 -1975.832,E2 -1975.832} C_VEL
LIN {X 0,Y 580.039,Z 667.023,A -85,B 0,C 180,E1 -1977.222,E2 -1977.222} C_VEL
LIN {X 0,Y 580.04,Z 668.456,A -85,B 0,C 180,E1 -1978.612,E2 -1978.612} C_VEL
LIN {X 0,Y 580.035,Z 668.996,A -85,B 0,C 180,E1 -1980,E2 -1980} C_VEL
LIN {X 0,Y 580.04,Z 668.516,A -85,B 0,C 180,E1 -1981.389,E2 -1981.389} C_VEL
LIN {X 0,Y 580.038,Z 667.143,A -85,B 0,C 180,E1 -1982.778,E2 -1982.778} C_VEL
LIN {X 0,Y 580.085,Z 664.732,A -85,B 0,C 180,E1 -1984.169,E2 -1984.169} C_VEL
LIN {X 0,Y 580.101,Z 660.331,A -85,B 0,C 180,E1 -1985.911,E2 -1985.911} C_VEL
LIN {X 0,Y 580.124,Z 655.628,A -85,B 0,C 180,E1 -1987.308,E2 -1987.308} C_VEL
LIN {X 0,Y 580.172,Z 649.695,A -85,B 0,C 180,E1 -1988.71,E2 -1988.71} C_VEL
LIN {X 0,Y 580.24,Z 641.541,A -85,B 0,C 180,E1 -1990.292,E2 -1990.292} C_VEL
LIN {X 0,Y 580.304,Z 632.767,A -85,B 0,C 180,E1 -1991.704,E2 -1991.704} C_VEL
LIN {X 0,Y 580.438,Z 622.28,A -85,B 0,C 180,E1 -1993.122,E2 -1993.122} C_VEL
LIN {X 0,Y 580.58,Z 610.764,A -85,B 0,C 180,E1 -1994.439,E2 -1994.439} C_VEL
LIN {X 0,Y 580.764,Z 598.621,A -85,B 0,C 180,E1 -1995.62,E2 -1995.62} C_VEL
LIN {X 0,Y 580.985,Z 585.629,A -85,B 0,C 180,E1 -1996.697,E2 -1996.697} C_VEL
LIN {X 0,Y 581.208,Z 571.558,A -85,B 0,C 180,E1 -1997.687,E2 -1997.687} C_VEL
LIN {X 0,Y 581.323,Z 564.775,A -85,B 0,C 180,E1 -1998.107,E2 -1998.107} C_VEL
LIN {X 0,Y 580.82,Z 559.772,A -85,B 0,C 180,E1 -1998.414,E2 -1998.414} C_VEL
LIN {X 0,Y 578.221,Z 551.753,A -85,B 0,C 180,E1 -1998.93,E2 -1998.93} C_VEL
LIN {X 0,Y 575.631,Z 543.549,A -85,B 0,C 180,E1 -1999.415,E2 -1999.415} C_VEL
LIN {X 0,Y 574.989,Z 538.259,A -85,B 0,C 180,E1 -1999.667,E2 -1999.667} C_VEL
LIN {X 0,Y 575.247,Z 521.399,A -85,B 0,C 180,E1 -2000.284,E2 -2000.284} C_VEL
LIN {X 0,Y 575.407,Z 506.376,A -85,B 0,C 180,E1 -2000.698,E2 -2000.698} C_VEL
LIN {X 0,Y 575.422,Z 493.193,A -85,B 0,C 180,E1 -2000.963,E2 -2000.963} C_VEL
